// Application/UserCode/MCU/MCU_VAR_1
VAR_GLOBAL
	(********************************************************)
	(*Rx*)
	(*MCUCommandResponse*)
	gu8_MCU_State						:	USINT;
	gu8_MCU_OperationalMode				:	USINT;
	gq_MCU_RegenDeratingStatus			:	BOOL;
	gu8_MCU_RegenDerating				:	USINT;
	gu8_MCU_TractionDerating			:	USINT;
	gu16_MCU_MaxMotorSpeedForward_Rx	:	UINT;
	gu16_MCU_MaxMotorSpeedReverse_Rx	:	UINT;
	gq_MCU_MaxMotorSpeedForwardStatus	:	BOOL;
	gq_MCU_MaxMotorSpeedReverseStatus	:	BOOL;
	gq_MCU_TractionDeratingStatus		:	BOOL;
	gu8_MCU_RollingCounter_Comm1		:	USINT;
	(*MCUCommandResponse2*)
	gu16_MCU_MotorSpeed_Rx				:	UINT;
	gu16_MCU_MotorAngle_Rx				:	UINT;
	gq_MVU_MotorAngleStatus				:	BOOL;
	gq_MCU_MotorSpeedStatus				:	BOOL;
	gq_MCU_SpeedReductionRequest		:	BOOL;
	gq_MCU_EmergencyStop				:	BOOL;
	gu8_MCU_RollingCounter_Comm2		:	USINT;
	(*MCUEventInfo1*)
	gq_MCU_Fault_PhaseToChassis					:	BOOL;
	gq_MCU_Fault_InterlockBatteryCable			:	BOOL;
	gq_MCU_Fault_InterlockMotorCable			:	BOOL;
	gq_MCU_Fault_DriveCoverWasOpened			:	BOOL;
	gq_MCU_Fault_PhaseToChassisStatus			:	BOOL;
	gq_MCU_Fault_InterlockBatteryCableStatus	:	BOOL;
	gq_MCU_Fault_InterlockMotorCableStatus		:	BOOL;
	gq_MCU_Fault_DriveCoverWasOpenedStatus		:	BOOL;
	(*MCUInfo1*)
	gu8_MCU_AuxiliaryVoltage_Rx					:	USINT;
	gu16_MCU_HighPowerVoltage					:	UINT;
	gq_MCU_HighPowerCurrentStatus				:	BOOL;
	gq_MCU_AuxiliaryVoltageStatus				:	BOOL;
	gq_MCU_HighPowerVoltageStatus				:	BOOL;
	gu16_MCU_HighPowerCurrent_Rx				:	UINT;
	gu8_MCU_RollingCounter_Info1				:	USINT;
	(*MCUInfo2*)
	gu16_MCU_MotorTorqueEstimated_Rx			:	UINT;
	gu16_MCU_TractionTorqueAvailable_Rx			:	UINT;
	gu16_MCU_RegenTorqueAvailable_Rx			:	UINT;
	gq_MCU_MotorTorqueEstimatedStatus			:	BOOL;
	gq_MCU_TractionTorqueAvailableStatus		:	BOOL;
	gq_MCU_RegenTorqueAvailableStatus			:	BOOL;
	gu8_MCU_RollingCounter_Info2				:	USINT;
	(*MCUOnEventInfo1*)
	gu16_MCU_EventID							:	UINT;
	gu8_MCU_RollingCounter_OnEventInfo1			:	USINT;
	(*MCUThermal1*)
	gu8_MCU_DriveCoolingFlowRequest_Rx			:	USINT;
	gu8_MCU_MotorCoolingFlowRequest_Rx			:	USINT;
	gu8_MCU_ThermalIndicator_Rx					:	USINT;
	gq_MCU_DriveCoolingFlowRequestStatus		:	BOOL;
	gq_MCU_MotorCoolingFlowRequestStatus		:	BOOL;
	gq_MCU_ThermalIndicatorStatus				:	BOOL;
	gu8_MCU_RollingCounter_Thermal1				:	USINT;
	(*MCUPollingMCUResponse*)
	gq_MCU_ResponseAcknowledgement				:	BOOL;
	gu8_MCU_MCUPollResponse_Multiplex			:	USINT;
		(*MCU MaxMotorSpeed*)
		gu16_MCU_MaxMotorSpeed_Rx				:	UINT;
		(*MCU MaxMotorTorque*)
		gu16_MCU_MaxMotorTorque_Rx				:	UINT;
		(*MCU ProtocolVersion*)
		gu8_MCU_MajorMCUProtocol				:	USINT;
		gu8_MCU_MinorMCUProtocol				:	USINT;
		gu8_MCU_ExtensionMajor					:	USINT;
		gu8_MCU_ExtensionMinor					:	USINT;
		(*MCU SWVersion1*)
		gu8_MCU_MajorMCUSW						:	USINT;
		gu8_MCU_MinorMCUSW						:	USINT;
		gu16_MCU_BranchMCUSW					:	UINT;
		(*MCU SWVersion2*)
		gu32_MCU_RevisionMCUSW					:	UDINT;
		(*MCU TotalMotorRotation*)
		gu32_MCU_TotalMotorRotation_LSB			:	UDINT;
		gu32_MCU_TotalMotorRotation_MSB			:	UDINT;
		gr_MCU_TotalMotorRotation_LSB			:	REAL;
		gr_MCU_TotalMotorRotation_MSB			:	REAL;
		gr_MCU_TotalMotorRotation				:	REAL;
		;
		(*MCUPollingVMU*)
		gu8_MCU_VMUBootNumber						:	USINT;
		(*VMUBootNumber*)
		gu16_MCU_BootNumber						:	UINT;
	
	(***************************************************************)
	(*Rx Conversion*)
	gr_MCU_MaxMotorSpeedForward		:	REAL;
	gr_MCU_MaxMotorSpeedReverse		:	REAL;
	gr_MCU_MotorSpeed				:	REAL;
	gr_MCU_MotorAngle				:	REAL;
	gr_MCU_AuxiliaryVoltage			:	REAL;
	gr_MCU_HighPowerCurrent			:	REAL;
	gr_MCU_MotorTorqueEstimated		:	REAL;
	gr_MCU_TractionTorqueAvailable	:	REAL;
	gr_MCU_RegenTorqueAvailable		:	REAL;
	gr_MCU_DriveCoolingFlowRequest	:	REAL;
	gr_MCU_MotorCoolingFlowRequest	:	REAL;
	gr_MCU_ThermalIndicator			:	REAL;
	gr_MCU_MaxMotorSpeed			:	REAL;
	gr_MCU_MaxMotorTorque			:	REAL;
	(****************************************************************)
	(*Tx*)
	(*VMU Comm1*)
	gu16_MCU_MaxChargeCurrent		:	UINT;
	gu8_MCU_OperationRequest		:	USINT;
	gu16_MCU_MaxDischargeCurrent	:	UINT;
	gu16_MCU_MaxBatteryVoltage		:	UINT;
	gq_MCU_MaxDiscahrgeCurrentStatus	:	BOOL;
	gq_MCU_MaxBatteryVoltageStatus	:	BOOL;
	gq_MCU_MinBatteryVoltageStatus	:	BOOL;
	gq_MCU_MaxChargeCurrentStatus	:	BOOL;
	gu16_MCU_MinBatteryVoltage		:	UINT;
	gu8_MCU_RollingCounter_VMUComm1	:	USINT;
	(*VMU Comm2*)
	gu8_MCU_OperationalMode_Tx		:	USINT;
	gu8_MCU_CommandMode				:	USINT;
	gq_MCU_SpeedCommandStatus		:	BOOL;
	gq_MCU_TorqueCommandStatus		:	BOOL;
	gu16_MCU_TorqueCommand_Tx		:	UINT;
	gu16_MCU_SpeedCommand_Tx		:	UINT;
	gu8_MCU_RollingCounter_VMUComm2	:	USINT;
	(*VMU CommandSafety*)
	gu16_MCU_ReferenceTorqueCommand_Tx	:	UINT;
	gu16_MCU_ReferenceSpeedCommand_Tx	:	UINT;
	gu8_MCU_ReferenceCommandMode		:	USINT;
	gu8_MCU_RollingCounter_VMUCommSafety	:	USINT;
	(*VMUPollingMCU*)
	gu8_MCU_VMUPollMCU_Multiplex	:	USINT;
		(*MCUMaxMotorSpeed*)
		gu16_MCU_MaxMotorSpeed_Tx	:	UINT;
		(*MCUMaxMotorTorque*)
		gu16_MCU_MaxMotorTorque_Tx	:	UINT;
		(*MCUProtocolVersion*)
		gu8_MCU_MajorMCUProtocol_Tx	:	USINT;
		gu8_MCU_MinorMCUProtocol_Tx	:	USINT;
		(*MCUSWVersion1*)
		gu8_MCU_MajorMCUSW_Tx			:	USINT;
		gu8_MCU_MinorMCUSW_Tx			:	USINT;
		gu16_MCU_BranchMCUSW_Tx			:	UINT;
		(*MCUSWVersion2*)
		gu32_MCU_RevisionMCUSW_Tx		:	UDINT;
		(*MCUTotalMotorRotation*)
		gu32_MCU_TotalMotorRotation_LSB_Tx	:	UDINT;
		gu32_MCU_TotalMotorRotation_MSB_Tx	:	UDINT;
	(*VMUPollingVMUResponse*)
	gq_MCU_PollVMUResponse_Acknowledgement	:	BOOL;
	gu8_MCU_PollVMUResponse_Multiplex		:	USINT;
		(*BootNumber*)
		gu16_MCU_BootNumber_Tx			:	UINT;		
	(*VMUSelectProtocolVersion*)
	gu8_MCU_SelectMajorMCUProtocol_Tx		:	USINT;
	gu8_MCU_SelectMinorMCUProtocol_Tx		:	USINT;
	
	(****************************************************************)
	(*True values - pre Tx*)
	gr_MCU_TorqueCommand_PreCF			:	REAL;
	gr_MCU_TorqueCommand_PreCF_Limited	:	REAL;
	gr_MCU_SpeedCommand_PreCF			:	REAL;
	gr_MCU_ReferenceTorqueCommand_PreCF	:	REAL;
	gr_MCU_ReferenceSpeedCommand_PreCF	:	REAL;
	gr_MCU_MaxMotorSpeed_PreCF			:	REAL;
	
	(****************************************************************)
	(*Latching Gear Selection*)
	gq_Gear_Neutral						:	BOOL;
	gq_Gear_Drive						:	BOOL;
	gq_Gear_DriveCrawl					:	BOOL;
	gq_Gear_Reverse						:	BOOL;
	gq_Gear_ReverseCrawl				:	BOOL;
	
	gq_MCU_CommsLoss					:	BOOL;
	
	(*Drivability*)
	gq_ABS_TorqueDisable				:	BOOL;
	
	gr_RearAxle_RelativeSpeed_kph		:	REAL;
	gu8_TractionLoss					:	USINT;
	gr_LeftWheels_RelativeSpeed_kph		:	REAL;
	gr_RightWheels_RelativeSpeed_kph	:	REAL;
	gu8_StabilityLoss					:	USINT;
	gq_ZeroTorqueRq						:	BOOL;
	gton_TorqueReIntro_Timer			:	TON;
	
	gr_RegenSOCMultiplier				:	REAL;
	gr_RegenMultiplierRq				:	REAL;
	gr_RegenIntroCF						:	REAL;
	gq_RegenActive						:	BOOL;
	gr_RegenSpeedDegrading				:	REAL;
	
	
	gr_VehicleTripDistance				:	REAL;
	gr_VehicleInitialTripDistance		:	REAL;
	
	gr_TorqueReIntro					:	REAL;
	gr_TorqueReIntroMax					:	REAL;
	
	gr_MCU_TorqueCommand_Limited	:	REAL;
	gr_MCU_PreviousTorqueCommand	:	REAL;
	
	gq_InitialProtocolGrab			:	BOOL;
END_VAR
VAR_GLOBAL CONSTANT
	MAXMOTORSPEED				:	USINT	:=	2;
	MAXMOTORTORQUE				:	USINT	:=	1;
	PROTOCOLVERSION				:	USINT	:=	0;
	SWVERSION1					:	USINT	:=	3;
	SWVERSION2					:	USINT	:=	4;
	TOTALMOTORROTATION			:	USINT	:=	5;
	TOTALMOTORROTATIONUSINTMCU	:	USINT	:=	6;
	
	VMUBOOTNUMBER				:	USINT	:=	0;
END_VAR

// Application/UserCode/Sevcon_Compressor/Sevcon2_VAR
VAR_GLOBAL
	(*********************************************************)
	
	(*Transmit*)
	(*Torque Demands 1*)
	gu16_Sevcon2_TorqueRq_Tx				:	UINT;
	gu16_Sevcon2_Controlword				:	UINT;
	gu16_Sevcon2_TorqueTractionLimit_Tx		:	UINT;
	gu8_Sevcon2_SEQCommand1					:	USINT;
	gu8_Sevcon2_CSCommand1					:	USINT;
	
	(*Torque Demands 2*)
	gu16_Sevcon2_TorqueRegenLimit_Tx		:	UINT;
	gu16_Sevcon2_SpeedLimitForward			:	UINT;
	gs16_Sevcon2_SpeedLimitReverse			:	INT;
	gu8_Sevcon2_SEQCommand2					:	USINT;
	gu8_Sevcon2_CSCommand2					:	USINT;
	
	(*Battery Demands*)
	gu16_Sevcon2_DCLink_ImaxDischarge		:	UINT;
	gs16_Sevcon2_DCLink_ImaxRecharge		:	INT;
	gu16_Sevcon2_DCLink_VoltageTarget_Tx	:	UINT;
	gu8_Sevcon2_SEQCurrentLimits			:	USINT;
	gu8_Sevcon2_CSCurrentLimits				:	USINT;
	
	(*I Demand Control*)
	gu16_Sevcon2_DebugIqDirectControl_Tx	:	UINT;
	gu16_Sevcon2_DebugIdDirectControl_Tx	:	UINT;
	gu8_Sevcon2_DirectCurrents				:	USINT;
	gu8_Sevcon2_CSDirectCurrents			:	USINT;
	
	(*********************************************************)
	
	(*Receive*)
	(*Torque Status 1*)
	gs16_Sevcon2_TorqueMeasured_Rx		:	INT;
	gs16_Sevcon2_SpeedMeasured			:	INT;
	gs16_Sevcon2_DCLink_Current			:	INT;
	gu8_Sevcon2_SEQ_Torque				:	USINT;
	gu8_Sevcon2_CS_Torque				:	USINT;
	
	(*Torque Status 2*)
	gs16_Sevcon2_TorqueAvailableForward_Rx	:	INT;
	gs16_Sevcon2_TorqueAvailableReverse_Rx	:	INT;
	gu8_Sevcon2_InverterStatus			:	USINT;
	gu8_Sevcon2_TorqueLimitCode			:	USINT;
	gu8_Sevcon2_SEQ_Status				:	USINT;
	gu8_Sevcon2_CS_Status				:	USINT;
	
	(*Temperature*)
	gs16_Sevcon2_TempRemaining			:	INT;
	gs16_Sevcon2_MotorTemp				:	INT;
	gs16_Sevcon2_DCLink_Voltage_Rx		:	INT;
	gu8_Sevcon2_SEQ_Temp					:	USINT;
	gu8_Sevcon2_CS_Temp					:	USINT;
	
	(**)
	gs16_Sevcon2_FaultCode				:	INT;
	gs32_Sevcon2_FaultData				:	DINT;
	gu8_Sevcon2_SEQ_Fault				:	USINT;
	gu8_Sevcon2_CS_Fault					:	USINT;
	
	(**)
	gs32_Sevcon2_EncoderPosition_Rx		:	DINT;
	
	(**)
	gs16_Sevcon2_Debug_Id_Act_Rx			:	INT;
	gs16_Sevcon2_Debug_Iq_Act_Rx			:	INT;
	gs16_Sevcon2_Debug_Id_Ref_Rx			:	INT;
	gs16_Sevcon2_Debug_Iq_Ref_Rx			:	INT;
	
	(**)
	gu8_Sevcon2_Debug_Temp_Junction0		:	USINT;
	gu8_Sevcon2_Debug_Temp_Junction1		:	USINT;
	gu8_Sevcon2_Debug_Temp_Junction2		:	USINT;
	gu8_Sevcon2_Debug_Temp_Junction3		:	USINT;
	gu8_Sevcon2_Debug_Temp_Junction4		:	USINT;
	gu8_Sevcon2_Debug_Temp_Junction5		:	USINT;
	gu8_Sevcon2_Debug_Temp_MotorMeasured	:	USINT;
	gu8_Sevcon2_Debug_Temp_MotorEstimate	:	USINT;
	
	(**)
	gu8_Sevcon2_Debug_Temp_CapEstimateFast	:	USINT;
	gu8_Sevcon2_Debug_Temp_Track				:	USINT;
	gu8_Sevcon2_Debug_Temp_CapEstimateSlow	:	USINT;
	gu8_Sevcon2_Debug_Temp_Heatsink			:	USINT;
	gu8_Sevcon2_Debug_Temp_DeltaTj			:	USINT;
	gu8_Sevcon2_Debug_Temp_Normalised		:	USINT;
	gu8_Sevcon2_Debug_Temp_Coolant			:	USINT;
	gu8_Sevcon2_Debug_Temp_Winding			:	USINT;
	
	(**)
	gs16_Sevcon2_Debug_MaxFlux				:	INT;
	gs16_Sevcon2_Debug_IvLim					:	INT;
	gs16_Sevcon2_Debug_IqMax					:	INT;
	gs16_Sevcon2_Debug_Ls_Rx					:	INT;
	
	(**)
	gs16_Sevcon2_Debug_Slip_Rx				:	INT;
	gs16_Sevcon2_Debug_LmSat_Rx				:	INT;
	gs16_Sevcon2_Debug_IqMax2				:	INT;
	gs16_Sevcon2_Debug_RecipFlux				:	INT;
	
	(*********************************************************)
	(*Tx conversion*)
	gr_Sevcon2_TorqueRq					:	REAL;
	gr_Sevcon2_TorqueTractionLimit		:	REAL;
	gr_Sevcon2_TorqueRegenLimit			:	REAL;
	gr_Sevcon2_DCLink_VoltageTarget		:	REAL;
	gr_Sevcon2_DebugIqDirectControl		:	REAL;
	gr_Sevcon2_DebugIdDirectControl		:	REAL;
	
	(*********************************************************)
	(*Rx converison*)
	gr_Sevcon2_TorqueMeasured			:	REAL;
	gr_Sevcon2_TorqueAvailableForward	:	REAL;
	gr_Sevcon2_TorqueAvailableReverse	:	REAL;
	gr_Sevcon2_DCLink_Voltage			:	REAL;
	gr_Sevcon2_EncoderPosition			:	REAL;
	gr_Sevcon2_Debug_Id_Act				:	REAL;
	gr_Sevcon2_Debug_Iq_Act				:	REAL;
	gr_Sevcon2_Debug_Id_Ref				:	REAL;
	gr_Sevcon2_Debug_Iq_Ref				:	REAL;
	gr_Sevcon2_Debug_Ls					:	REAL;
	gr_Sevcon2_Debug_Slip				:	REAL;
	gr_Sevcon2_Debug_LmSat				:	REAL;
	
	
	gq_Sevcon2_CommsLoss				:	BOOL;
	
END_VAR

// Application/UserCode/Sevcon_Compressor/Sevcon2_VAR_1
VAR_GLOBAL
	(*********************************************************)
	
	(*Transmit*)
	(*Torque Demands 1*)
	gu16_Sevcon2_TorqueRq_Tx				:	UINT;
	gu16_Sevcon2_Controlword				:	UINT;
	gu16_Sevcon2_TorqueTractionLimit_Tx		:	UINT;
	gu8_Sevcon2_SEQCommand1					:	USINT;
	gu8_Sevcon2_CSCommand1					:	USINT;
	
	(*Torque Demands 2*)
	gu16_Sevcon2_TorqueRegenLimit_Tx		:	UINT;
	gu16_Sevcon2_SpeedLimitForward			:	UINT;
	gs16_Sevcon2_SpeedLimitReverse			:	INT;
	gu8_Sevcon2_SEQCommand2					:	USINT;
	gu8_Sevcon2_CSCommand2					:	USINT;
	
	(*Battery Demands*)
	gu16_Sevcon2_DCLink_ImaxDischarge		:	UINT;
	gs16_Sevcon2_DCLink_ImaxRecharge		:	INT;
	gu16_Sevcon2_DCLink_VoltageTarget_Tx	:	UINT;
	gu8_Sevcon2_SEQCurrentLimits			:	USINT;
	gu8_Sevcon2_CSCurrentLimits				:	USINT;
	
	(*I Demand Control*)
	gu16_Sevcon2_DebugIqDirectControl_Tx	:	UINT;
	gu16_Sevcon2_DebugIdDirectControl_Tx	:	UINT;
	gu8_Sevcon2_DirectCurrents				:	USINT;
	gu8_Sevcon2_CSDirectCurrents			:	USINT;
	
	(*********************************************************)
	
	(*Receive*)
	(*Torque Status 1*)
	gs16_Sevcon2_TorqueMeasured_Rx		:	INT;
	gs16_Sevcon2_SpeedMeasured			:	INT;
	gs16_Sevcon2_DCLink_Current			:	INT;
	gu8_Sevcon2_SEQ_Torque				:	USINT;
	gu8_Sevcon2_CS_Torque				:	USINT;
	
	(*Torque Status 2*)
	gs16_Sevcon2_TorqueAvailableForward_Rx	:	INT;
	gs16_Sevcon2_TorqueAvailableReverse_Rx	:	INT;
	gu8_Sevcon2_InverterStatus			:	USINT;
	gu8_Sevcon2_TorqueLimitCode			:	USINT;
	gu8_Sevcon2_SEQ_Status				:	USINT;
	gu8_Sevcon2_CS_Status				:	USINT;
	
	(*Temperature*)
	gs16_Sevcon2_TempRemaining			:	INT;
	gs16_Sevcon2_MotorTemp				:	INT;
	gs16_Sevcon2_DCLink_Voltage_Rx		:	INT;
	gu8_Sevcon2_SEQ_Temp					:	USINT;
	gu8_Sevcon2_CS_Temp					:	USINT;
	
	(**)
	gs16_Sevcon2_FaultCode				:	INT;
	gs32_Sevcon2_FaultData				:	DINT;
	gu8_Sevcon2_SEQ_Fault				:	USINT;
	gu8_Sevcon2_CS_Fault					:	USINT;
	
	(**)
	gs32_Sevcon2_EncoderPosition_Rx		:	DINT;
	
	(**)
	gs16_Sevcon2_Debug_Id_Act_Rx			:	INT;
	gs16_Sevcon2_Debug_Iq_Act_Rx			:	INT;
	gs16_Sevcon2_Debug_Id_Ref_Rx			:	INT;
	gs16_Sevcon2_Debug_Iq_Ref_Rx			:	INT;
	
	(**)
	gu8_Sevcon2_Debug_Temp_Junction0		:	USINT;
	gu8_Sevcon2_Debug_Temp_Junction1		:	USINT;
	gu8_Sevcon2_Debug_Temp_Junction2		:	USINT;
	gu8_Sevcon2_Debug_Temp_Junction3		:	USINT;
	gu8_Sevcon2_Debug_Temp_Junction4		:	USINT;
	gu8_Sevcon2_Debug_Temp_Junction5		:	USINT;
	gu8_Sevcon2_Debug_Temp_MotorMeasured	:	USINT;
	gu8_Sevcon2_Debug_Temp_MotorEstimate	:	USINT;
	
	(**)
	gu8_Sevcon2_Debug_Temp_CapEstimateFast	:	USINT;
	gu8_Sevcon2_Debug_Temp_Track				:	USINT;
	gu8_Sevcon2_Debug_Temp_CapEstimateSlow	:	USINT;
	gu8_Sevcon2_Debug_Temp_Heatsink			:	USINT;
	gu8_Sevcon2_Debug_Temp_DeltaTj			:	USINT;
	gu8_Sevcon2_Debug_Temp_Normalised		:	USINT;
	gu8_Sevcon2_Debug_Temp_Coolant			:	USINT;
	gu8_Sevcon2_Debug_Temp_Winding			:	USINT;
	
	(**)
	gs16_Sevcon2_Debug_MaxFlux				:	INT;
	gs16_Sevcon2_Debug_IvLim					:	INT;
	gs16_Sevcon2_Debug_IqMax					:	INT;
	gs16_Sevcon2_Debug_Ls_Rx					:	INT;
	
	(**)
	gs16_Sevcon2_Debug_Slip_Rx				:	INT;
	gs16_Sevcon2_Debug_LmSat_Rx				:	INT;
	gs16_Sevcon2_Debug_IqMax2				:	INT;
	gs16_Sevcon2_Debug_RecipFlux				:	INT;
	
	(*********************************************************)
	(*Tx conversion*)
	gr_Sevcon2_TorqueRq					:	REAL;
	gr_Sevcon2_TorqueTractionLimit		:	REAL;
	gr_Sevcon2_TorqueRegenLimit			:	REAL;
	gr_Sevcon2_DCLink_VoltageTarget		:	REAL;
	gr_Sevcon2_DebugIqDirectControl		:	REAL;
	gr_Sevcon2_DebugIdDirectControl		:	REAL;
	
	(*********************************************************)
	(*Rx converison*)
	gr_Sevcon2_TorqueMeasured			:	REAL;
	gr_Sevcon2_TorqueAvailableForward	:	REAL;
	gr_Sevcon2_TorqueAvailableReverse	:	REAL;
	gr_Sevcon2_DCLink_Voltage			:	REAL;
	gr_Sevcon2_EncoderPosition			:	REAL;
	gr_Sevcon2_Debug_Id_Act				:	REAL;
	gr_Sevcon2_Debug_Iq_Act				:	REAL;
	gr_Sevcon2_Debug_Id_Ref				:	REAL;
	gr_Sevcon2_Debug_Iq_Ref				:	REAL;
	gr_Sevcon2_Debug_Ls					:	REAL;
	gr_Sevcon2_Debug_Slip				:	REAL;
	gr_Sevcon2_Debug_LmSat				:	REAL;
	
	
	gq_Sevcon2_CommsLoss				:	BOOL;
	
END_VAR

// Application/UserCode/Sevcon ePTO/Sevcon_ePTO_VAR
VAR_GLOBAL
	(*********************************************************)
	
	(*Transmit*)
	(*Torque Demands 1*)
	gu16_Sevcon_ePTO_TorqueRq_Tx				:	UINT;
	gu16_Sevcon_ePTO_Controlword				:	UINT;
	gu16_Sevcon_ePTO_TorqueTractionLimit_Tx		:	UINT;
	gu8_Sevcon_ePTO_SEQCommand1					:	USINT;
	gu8_Sevcon_ePTO_CSCommand1					:	USINT;
	
	(*Torque Demands 2*)
	gu16_Sevcon_ePTO_TorqueRegenLimit_Tx		:	UINT;
	gu16_Sevcon_ePTO_SpeedLimitForward			:	UINT;
	gs16_Sevcon_ePTO_SpeedLimitReverse			:	INT;
	gu8_Sevcon_ePTO_SEQCommand2					:	USINT;
	gu8_Sevcon_ePTO_CSCommand2					:	USINT;
	
	(*Battery Demands*)
	gu16_Sevcon_ePTO_DCLink_ImaxDischarge		:	UINT;
	gs16_Sevcon_ePTO_DCLink_ImaxRecharge		:	INT;
	gu16_Sevcon_ePTO_DCLink_VoltageTarget_Tx	:	UINT;
	gu8_Sevcon_ePTO_SEQCurrentLimits			:	USINT;
	gu8_Sevcon_ePTO_CSCurrentLimits				:	USINT;
	
	(*I Demand Control*)
	gu16_Sevcon_ePTO_DebugIqDirectControl_Tx	:	UINT;
	gu16_Sevcon_ePTO_DebugIdDirectControl_Tx	:	UINT;
	gu8_Sevcon_ePTO_DirectCurrents				:	USINT;
	gu8_Sevcon_ePTO_CSDirectCurrents			:	USINT;
	
	(*********************************************************)
	
	(*Receive*)
	(*Torque Status 1*)
	gs16_Sevcon_ePTO_TorqueMeasured_Rx		:	INT;
	gs16_Sevcon_ePTO_SpeedMeasured			:	INT;
	gs16_Sevcon_ePTO_DCLink_Current			:	INT;
	gu8_Sevcon_ePTO_SEQ_Torque				:	USINT;
	gu8_Sevcon_ePTO_CS_Torque				:	USINT;
	
	(*Torque Status 2*)
	gs16_Sevcon_ePTO_TorqueAvailableForward_Rx	:	INT;
	gs16_Sevcon_ePTO_TorqueAvailableReverse_Rx	:	INT;
	gu8_Sevcon_ePTO_InverterStatus			:	USINT;
	gu8_Sevcon_ePTO_TorqueLimitCode			:	USINT;
	gu8_Sevcon_ePTO_SEQ_Status				:	USINT;
	gu8_Sevcon_ePTO_CS_Status				:	USINT;
	
	(*Temperature*)
	gs16_Sevcon_ePTO_TempRemaining			:	INT;
	gs16_Sevcon_ePTO_MotorTemp				:	INT;
	gs16_Sevcon_ePTO_DCLink_Voltage_Rx		:	INT;
	gu8_Sevcon_ePTO_SEQ_Temp					:	USINT;
	gu8_Sevcon_ePTO_CS_Temp					:	USINT;
	
	(**)
	gs16_Sevcon_ePTO_FaultCode				:	INT;
	gs32_Sevcon_ePTO_FaultData				:	DINT;
	gu8_Sevcon_ePTO_SEQ_Fault				:	USINT;
	gu8_Sevcon_ePTO_CS_Fault					:	USINT;
	
	(**)
	gs32_Sevcon_ePTO_EncoderPosition_Rx		:	DINT;
	
	(**)
	gs16_Sevcon_ePTO_Debug_Id_Act_Rx			:	INT;
	gs16_Sevcon_ePTO_Debug_Iq_Act_Rx			:	INT;
	gs16_Sevcon_ePTO_Debug_Id_Ref_Rx			:	INT;
	gs16_Sevcon_ePTO_Debug_Iq_Ref_Rx			:	INT;
	
	(**)
	gu8_Sevcon_ePTO_Debug_Temp_Junction0		:	USINT;
	gu8_Sevcon_ePTO_Debug_Temp_Junction1		:	USINT;
	gu8_Sevcon_ePTO_Debug_Temp_Junction2		:	USINT;
	gu8_Sevcon_ePTO_Debug_Temp_Junction3		:	USINT;
	gu8_Sevcon_ePTO_Debug_Temp_Junction4		:	USINT;
	gu8_Sevcon_ePTO_Debug_Temp_Junction5		:	USINT;
	gu8_Sevcon_ePTO_Debug_Temp_MotorMeasured	:	USINT;
	gu8_Sevcon_ePTO_Debug_Temp_MotorEstimate	:	USINT;
	
	(**)
	gu8_Sevcon_ePTO_Debug_Temp_CapEstimateFast	:	USINT;
	gu8_Sevcon_ePTO_Debug_Temp_Track				:	USINT;
	gu8_Sevcon_ePTO_Debug_Temp_CapEstimateSlow	:	USINT;
	gu8_Sevcon_ePTO_Debug_Temp_Heatsink			:	USINT;
	gu8_Sevcon_ePTO_Debug_Temp_DeltaTj			:	USINT;
	gu8_Sevcon_ePTO_Debug_Temp_Normalised		:	USINT;
	gu8_Sevcon_ePTO_Debug_Temp_Coolant			:	USINT;
	gu8_Sevcon_ePTO_Debug_Temp_Winding			:	USINT;
	
	(**)
	gs16_Sevcon_ePTO_Debug_MaxFlux				:	INT;
	gs16_Sevcon_ePTO_Debug_IvLim					:	INT;
	gs16_Sevcon_ePTO_Debug_IqMax					:	INT;
	gs16_Sevcon_ePTO_Debug_Ls_Rx					:	INT;
	
	(**)
	gs16_Sevcon_ePTO_Debug_Slip_Rx				:	INT;
	gs16_Sevcon_ePTO_Debug_LmSat_Rx				:	INT;
	gs16_Sevcon_ePTO_Debug_IqMax2				:	INT;
	gs16_Sevcon_ePTO_Debug_RecipFlux				:	INT;
	
	(*********************************************************)
	(*Tx conversion*)
	gr_Sevcon_ePTO_TorqueRq					:	REAL;
	gr_Sevcon_ePTO_TorqueTractionLimit		:	REAL;
	gr_Sevcon_ePTO_TorqueRegenLimit			:	REAL;
	gr_Sevcon_ePTO_DCLink_VoltageTarget		:	REAL;
	gr_Sevcon_ePTO_DebugIqDirectControl		:	REAL;
	gr_Sevcon_ePTO_DebugIdDirectControl		:	REAL;
	
	(*********************************************************)
	(*Rx converison*)
	gr_Sevcon_ePTO_TorqueMeasured			:	REAL;
	gr_Sevcon_ePTO_TorqueAvailableForward	:	REAL;
	gr_Sevcon_ePTO_TorqueAvailableReverse	:	REAL;
	gr_Sevcon_ePTO_DCLink_Voltage			:	REAL;
	gr_Sevcon_ePTO_EncoderPosition			:	REAL;
	gr_Sevcon_ePTO_Debug_Id_Act				:	REAL;
	gr_Sevcon_ePTO_Debug_Iq_Act				:	REAL;
	gr_Sevcon_ePTO_Debug_Id_Ref				:	REAL;
	gr_Sevcon_ePTO_Debug_Iq_Ref				:	REAL;
	gr_Sevcon_ePTO_Debug_Ls					:	REAL;
	gr_Sevcon_ePTO_Debug_Slip				:	REAL;
	gr_Sevcon_ePTO_Debug_LmSat				:	REAL;
	
	
	
	
END_VAR

// Application/UserCode/Sevcon_PSP/Sevcon_Steer_VAR_1
VAR_GLOBAL
	(*********************************************************)
	
	(*Transmit*)
	(*Torque Demands 1*)
	gu16_Sevcon1_TorqueRq_Tx				:	UINT;
	gu16_Sevcon1_Controlword				:	UINT;
	gu16_Sevcon1_TorqueTractionLimit_Tx		:	UINT;
	gu8_Sevcon1_SEQCommand1					:	USINT;
	gu8_Sevcon1_CSCommand1					:	USINT;
	
	(*Torque Demands 2*)
	gu16_Sevcon1_TorqueRegenLimit_Tx		:	UINT;
	gu16_Sevcon1_SpeedLimitForward			:	UINT;
	gs16_Sevcon1_SpeedLimitReverse			:	INT;
	gu8_Sevcon1_SEQCommand2					:	USINT;
	gu8_Sevcon1_CSCommand2					:	USINT;
	
	(*Battery Demands*)
	gu16_Sevcon1_DCLink_ImaxDischarge		:	UINT;
	gs16_Sevcon1_DCLink_ImaxRecharge		:	INT;
	gu16_Sevcon1_DCLink_VoltageTarget_Tx	:	UINT;
	gu8_Sevcon1_SEQCurrentLimits			:	USINT;
	gu8_Sevcon1_CSCurrentLimits				:	USINT;
	
	(*I Demand Control*)
	gu16_Sevcon1_DebugIqDirectControl_Tx	:	UINT;
	gu16_Sevcon1_DebugIdDirectControl_Tx	:	UINT;
	gu8_Sevcon1_DirectCurrents				:	USINT;
	gu8_Sevcon1_CSDirectCurrents			:	USINT;
	
	(*********************************************************)
	
	(*Receive*)
	(*Torque Status 1*)
	gs16_Sevcon1_TorqueMeasured_Rx		:	INT;
	gs16_Sevcon1_SpeedMeasured			:	INT;
	gs16_Sevcon1_DCLink_Current			:	INT;
	gu8_Sevcon1_SEQ_Torque				:	USINT;
	gu8_Sevcon1_CS_Torque				:	USINT;
	
	(*Torque Status 2*)
	gs16_Sevcon1_TorqueAvailableForward_Rx	:	INT;
	gs16_Sevcon1_TorqueAvailableReverse_Rx	:	INT;
	gu8_Sevcon1_InverterStatus			:	USINT;
	gu8_Sevcon1_TorqueLimitCode			:	USINT;
	gu8_Sevcon1_SEQ_Status				:	USINT;
	gu8_Sevcon1_CS_Status				:	USINT;
	
	(*Temperature*)
	gs16_Sevcon1_TempRemaining			:	INT;
	gs16_Sevcon1_MotorTemp				:	INT;
	gs16_Sevcon1_DCLink_Voltage_Rx		:	INT;
	gu8_Sevcon1_SEQ_Temp					:	USINT;
	gu8_Sevcon1_CS_Temp					:	USINT;
	
	(**)
	gs16_Sevcon1_FaultCode				:	INT;
	gs32_Sevcon1_FaultData				:	DINT;
	gu8_Sevcon1_SEQ_Fault				:	USINT;
	gu8_Sevcon1_CS_Fault					:	USINT;
	
	(**)
	gs32_Sevcon1_EncoderPosition_Rx		:	DINT;
	
	(**)
	gs16_Sevcon1_Debug_Id_Act_Rx			:	INT;
	gs16_Sevcon1_Debug_Iq_Act_Rx			:	INT;
	gs16_Sevcon1_Debug_Id_Ref_Rx			:	INT;
	gs16_Sevcon1_Debug_Iq_Ref_Rx			:	INT;
	
	(**)
	gu8_Sevcon1_Debug_Temp_Junction0		:	USINT;
	gu8_Sevcon1_Debug_Temp_Junction1		:	USINT;
	gu8_Sevcon1_Debug_Temp_Junction2		:	USINT;
	gu8_Sevcon1_Debug_Temp_Junction3		:	USINT;
	gu8_Sevcon1_Debug_Temp_Junction4		:	USINT;
	gu8_Sevcon1_Debug_Temp_Junction5		:	USINT;
	gu8_Sevcon1_Debug_Temp_MotorMeasured	:	USINT;
	gu8_Sevcon1_Debug_Temp_MotorEstimate	:	USINT;
	
	(**)
	gu8_Sevcon1_Debug_Temp_CapEstimateFast	:	USINT;
	gu8_Sevcon1_Debug_Temp_Track				:	USINT;
	gu8_Sevcon1_Debug_Temp_CapEstimateSlow	:	USINT;
	gu8_Sevcon1_Debug_Temp_Heatsink			:	USINT;
	gu8_Sevcon1_Debug_Temp_DeltaTj			:	USINT;
	gu8_Sevcon1_Debug_Temp_Normalised		:	USINT;
	gu8_Sevcon1_Debug_Temp_Coolant			:	USINT;
	gu8_Sevcon1_Debug_Temp_Winding			:	USINT;
	
	(**)
	gs16_Sevcon1_Debug_MaxFlux				:	INT;
	gs16_Sevcon1_Debug_IvLim					:	INT;
	gs16_Sevcon1_Debug_IqMax					:	INT;
	gs16_Sevcon1_Debug_Ls_Rx					:	INT;
	
	(**)
	gs16_Sevcon1_Debug_Slip_Rx				:	INT;
	gs16_Sevcon1_Debug_LmSat_Rx				:	INT;
	gs16_Sevcon1_Debug_IqMax2				:	INT;
	gs16_Sevcon1_Debug_RecipFlux				:	INT;
	
	(*********************************************************)
	(*Tx conversion*)
	gr_Sevcon1_TorqueRq					:	REAL;
	gr_Sevcon1_TorqueTractionLimit		:	REAL;
	gr_Sevcon1_TorqueRegenLimit			:	REAL;
	gr_Sevcon1_DCLink_VoltageTarget		:	REAL;
	gr_Sevcon1_DebugIqDirectControl		:	REAL;
	gr_Sevcon1_DebugIdDirectControl		:	REAL;
	
	(*********************************************************)
	(*Rx converison*)
	gr_Sevcon1_TorqueMeasured			:	REAL;
	gr_Sevcon1_TorqueAvailableForward	:	REAL;
	gr_Sevcon1_TorqueAvailableReverse	:	REAL;
	gr_Sevcon1_DCLink_Voltage			:	REAL;
	gr_Sevcon1_EncoderPosition			:	REAL;
	gr_Sevcon1_Debug_Id_Act				:	REAL;
	gr_Sevcon1_Debug_Iq_Act				:	REAL;
	gr_Sevcon1_Debug_Id_Ref				:	REAL;
	gr_Sevcon1_Debug_Iq_Ref				:	REAL;
	gr_Sevcon1_Debug_Ls					:	REAL;
	gr_Sevcon1_Debug_Slip				:	REAL;
	gr_Sevcon1_Debug_LmSat				:	REAL;
	
	
	gq_Sevcon1_CommsLoss				:	BOOL;
	
END_VAR

// Application/UserCode/UserMramUsage_1/UserMramVariables_1
VAR_GLOBAL
	///[Pointer to the start of the NVRAM area.]
	G_pUserMramStructure: POINTER TO UserMramStructure;
	///[Pointer to the start of the OD parameter image.]
	G_UserMramStructureDefault: UserMramStructure;
END_VAR

// Application/UserCode/UserMramUsage/UserMramVariables
VAR_GLOBAL
	///[Pointer to the start of the NVRAM area.]
	G_pUserMramStructure: POINTER TO UserMramStructure;
	///[Pointer to the start of the OD parameter image.]
	G_UserMramStructureDefault: UserMramStructure;
END_VAR

// Application/CodeTemplate/Globals/CANopen_CAN1/G_CAN1_VAR
///
///NOTE! NOTE! NOTE! NOTE! NOTE! NOTE! NOTE! NOTE! NOTE! NOTE! NOTE!
/// 	                    
/// This object is created by Epec MultiTool
/// User changes are overwritten when project is imported
///
/// Content
/// - CANopen OD index data
///
{attribute 'qualified_only'}
VAR_GLOBAL
	/// 16#1000 Information about the device type
	DeviceType_Device1: UDINT := 405;
	/// 16#1001 Error information
	ErrorReg_Device1: USINT := 0;
	/// 16#2128 PDO Dummy Variable Index
	CAN1_TPDO_DUMMY: BYTE := 0;
	/// 16#2129 PDO Dummy Variable Index
	CAN1_RPDO_DUMMY: BYTE := 0;
	/// 16#2131 Parameter CSV unique ID
	Parameter_CSV_unique_ID1: UINT := 16#0000;
END_VAR

// Application/CodeTemplate/Globals/CANopen_CAN1/G_CANopen_CAN1
///
///NOTE! NOTE! NOTE! NOTE! NOTE! NOTE! NOTE! NOTE! NOTE! NOTE! NOTE!
/// 	                    
/// This object is created by Epec MultiTool
/// User changes are overwritten when project is imported
///
/// Content
/// - CANopen protocol variable definitions
///
{attribute 'qualified_only'}
{attribute 'global_init_slot' := '49991'}
VAR_GLOBAL
	/// CAN device
	Device: EPEC_CANopen.Device;
	/// Object Dictionary data
	OD: EPEC_CANopen.OD;
	ODEntrys: ARRAY[1..74] OF EPEC_CANopen.ODEntry;
	/// Protocol data
	Protocols: ARRAY[1..5] OF EPEC_CANopen.ProtocolEntry;
	/// Heartbeat producer/consumer protocol data
	HB: EPEC_CANopen.HBData;
	/// Heartbeat producer/consumer protocol handler
	HB_Handler: EPEC_CANopen.CANopenHB;
	/// NMT protocol data
	NMT: EPEC_CANopen.NMTData;
	/// NMT protocol handler
	NMT_Handler: EPEC_CANopen.CANopenNMT;
	/// SDO server protocol data
	SSDO: EPEC_CANopen.SSDOData;
	/// SDO server protocol handler
	SSDO_Handler: EPEC_CANopen.CANopenSDOServer;
	/// GFC protocol data
	GFC: EPEC_CANopen.GFCData;
	/// GFC protocol handler
	GFC_Handler: EPEC_CANopen.CANopenGFC;
	/// SDO client instances
	CSDOS: ARRAY[1..127] OF EPEC_CANopen.CANopenCSDO := [];
	SaveAll: EPEC_ODSave.SaveODSaveAll;
	DeleteAll: EPEC_ODSave.SaveODDeleteAll;
	Initialize: EPEC_ODSave.SaveODInitialize;
	SaveData: ARRAY[0..3] OF EPEC_ODSave.SaveODSubIndexDescription := [(StartIndex := 16#1000, EndIndex := 16#FFFF, GroupNum := 1), (StartIndex := 16#1000, EndIndex := 16#1FFF, GroupNum := 1), (StartIndex := 16#2000, EndIndex := 16#FFFF, GroupNum := 1), (StartIndex := 16#0, EndIndex := 16#0, GroupNum := 1)];
	SaveSubData1010h: EPEC_ODSave.SaveODSubService;
END_VAR

// Application/CodeTemplate/Globals/CANopen_CAN1/G_CANopen_CAN1_VAR
///
///NOTE! NOTE! NOTE! NOTE! NOTE! NOTE! NOTE! NOTE! NOTE! NOTE! NOTE!
/// 	                    
/// This object is created by Epec MultiTool
/// User changes are overwritten when project is imported
///
/// Content
/// - 
/// 
{attribute 'qualified_only'}
{attribute 'global_init_slot' := '49990'}
VAR_GLOBAL
	OD_Error: EPEC_CANopen.Errors := EPEC_CANopen.Errors.NotInitialized;
	ODSave_Error: EPEC_ODSave.SaveODErrors;
	Callback_Error: EPEC_CANopen.Errors := EPEC_CANopen.Errors.NotInitialized;
	ProtocolAdded: ARRAY[1..5] OF BOOL := [5(0)];
	HB_Error: EPEC_CANopen.Errors := EPEC_CANopen.Errors.NotInitialized;
	NMT_Error: EPEC_CANopen.Errors := EPEC_CANopen.Errors.NotInitialized;
	SSDO_Error: EPEC_CANopen.Errors := EPEC_CANopen.Errors.NotInitialized;
	GFC_Error: EPEC_CANopen.Errors := EPEC_CANopen.Errors.NotInitialized;
	/// GFC status
	GFC_Status: BYTE;
	CSDO_Error: EPEC_CANopen.Errors := EPEC_CANopen.Errors.NotInitialized;
	SaveSigns1010: ARRAY[0..3] OF DWORD;
END_VAR

// Application/CodeTemplate/Globals/CANopen_CAN2/G_CAN2_VAR
///
///NOTE! NOTE! NOTE! NOTE! NOTE! NOTE! NOTE! NOTE! NOTE! NOTE! NOTE!
/// 	                    
/// This object is created by Epec MultiTool
/// User changes are overwritten when project is imported
///
/// Content
/// - CANopen OD index data
///
{attribute 'qualified_only'}
VAR_GLOBAL
	/// 16#1000 Information about the device type
	DeviceType_Device2: UDINT := 405;
	/// 16#1001 Error information
	ErrorReg_Device2: USINT := 0;
	/// 16#2128 PDO Dummy Variable Index
	CAN2_TPDO_DUMMY: BYTE := 0;
	/// 16#2129 PDO Dummy Variable Index
	CAN2_RPDO_DUMMY: BYTE := 0;
	/// 16#2131 Parameter CSV unique ID
	Parameter_CSV_unique_ID2: UINT := 16#0000;
END_VAR

// Application/CodeTemplate/Globals/CANopen_CAN2/G_CANopen_CAN2
///
///NOTE! NOTE! NOTE! NOTE! NOTE! NOTE! NOTE! NOTE! NOTE! NOTE! NOTE!
/// 	                    
/// This object is created by Epec MultiTool
/// User changes are overwritten when project is imported
///
/// Content
/// - CANopen protocol variable definitions
///
{attribute 'qualified_only'}
{attribute 'global_init_slot' := '49991'}
VAR_GLOBAL
	/// CAN device
	Device: EPEC_CANopen.Device;
	/// Object Dictionary data
	OD: EPEC_CANopen.OD;
	ODEntrys: ARRAY[1..66] OF EPEC_CANopen.ODEntry;
	/// Protocol data
	Protocols: ARRAY[1..5] OF EPEC_CANopen.ProtocolEntry;
	/// Heartbeat producer/consumer protocol data
	HB: EPEC_CANopen.HBData;
	/// Heartbeat producer/consumer protocol handler
	HB_Handler: EPEC_CANopen.CANopenHB;
	/// NMT protocol data
	NMT: EPEC_CANopen.NMTData;
	/// NMT protocol handler
	NMT_Handler: EPEC_CANopen.CANopenNMT;
	/// SDO server protocol data
	SSDO: EPEC_CANopen.SSDOData;
	/// SDO server protocol handler
	SSDO_Handler: EPEC_CANopen.CANopenSDOServer;
	/// GFC protocol data
	GFC: EPEC_CANopen.GFCData;
	/// GFC protocol handler
	GFC_Handler: EPEC_CANopen.CANopenGFC;
	/// SDO client instances
	CSDOS: ARRAY[1..127] OF EPEC_CANopen.CANopenCSDO := [];
	SaveAll: EPEC_ODSave.SaveODSaveAll;
	DeleteAll: EPEC_ODSave.SaveODDeleteAll;
	Initialize: EPEC_ODSave.SaveODInitialize;
	SaveData: ARRAY[0..3] OF EPEC_ODSave.SaveODSubIndexDescription := [(StartIndex := 16#1000, EndIndex := 16#FFFF, GroupNum := 2), (StartIndex := 16#1000, EndIndex := 16#1FFF, GroupNum := 2), (StartIndex := 16#2000, EndIndex := 16#FFFF, GroupNum := 2), (StartIndex := 16#0, EndIndex := 16#0, GroupNum := 2)];
	SaveSubData1010h: EPEC_ODSave.SaveODSubService;
END_VAR

// Application/CodeTemplate/Globals/CANopen_CAN2/G_CANopen_CAN2_VAR
///
///NOTE! NOTE! NOTE! NOTE! NOTE! NOTE! NOTE! NOTE! NOTE! NOTE! NOTE!
/// 	                    
/// This object is created by Epec MultiTool
/// User changes are overwritten when project is imported
///
/// Content
/// - 
/// 
{attribute 'qualified_only'}
{attribute 'global_init_slot' := '49990'}
VAR_GLOBAL
	OD_Error: EPEC_CANopen.Errors := EPEC_CANopen.Errors.NotInitialized;
	ODSave_Error: EPEC_ODSave.SaveODErrors;
	Callback_Error: EPEC_CANopen.Errors := EPEC_CANopen.Errors.NotInitialized;
	ProtocolAdded: ARRAY[1..5] OF BOOL := [5(0)];
	HB_Error: EPEC_CANopen.Errors := EPEC_CANopen.Errors.NotInitialized;
	NMT_Error: EPEC_CANopen.Errors := EPEC_CANopen.Errors.NotInitialized;
	SSDO_Error: EPEC_CANopen.Errors := EPEC_CANopen.Errors.NotInitialized;
	GFC_Error: EPEC_CANopen.Errors := EPEC_CANopen.Errors.NotInitialized;
	/// GFC status
	GFC_Status: BYTE;
	CSDO_Error: EPEC_CANopen.Errors := EPEC_CANopen.Errors.NotInitialized;
	SaveSigns1010: ARRAY[0..3] OF DWORD;
END_VAR

// Application/CodeTemplate/Globals/CANopen_CAN3/G_CAN3_VAR
///
///NOTE! NOTE! NOTE! NOTE! NOTE! NOTE! NOTE! NOTE! NOTE! NOTE! NOTE!
/// 	                    
/// This object is created by Epec MultiTool
/// User changes are overwritten when project is imported
///
/// Content
/// - CANopen OD index data
///
{attribute 'qualified_only'}
VAR_GLOBAL
	/// 16#1000 Information about the device type
	DeviceType_Device3: UDINT := 405;
	/// 16#1001 Error information
	ErrorReg_Device3: USINT := 0;
	/// 16#2129 PDO Dummy Variable Index
	CAN3_PDO_DUMMY: BYTE := 0;
	/// 16#2131 Parameter CSV unique ID
	Parameter_CSV_unique_ID3: UINT := 16#0000;
END_VAR

// Application/CodeTemplate/Globals/CANopen_CAN3/G_CANopen_CAN3
///
///NOTE! NOTE! NOTE! NOTE! NOTE! NOTE! NOTE! NOTE! NOTE! NOTE! NOTE!
/// 	                    
/// This object is created by Epec MultiTool
/// User changes are overwritten when project is imported
///
/// Content
/// - CANopen protocol variable definitions
///
{attribute 'qualified_only'}
{attribute 'global_init_slot' := '49991'}
VAR_GLOBAL
	/// CAN device
	Device: EPEC_CANopen.Device;
	/// Object Dictionary data
	OD: EPEC_CANopen.OD;
	ODEntrys: ARRAY[1..65] OF EPEC_CANopen.ODEntry;
	/// Protocol data
	Protocols: ARRAY[1..5] OF EPEC_CANopen.ProtocolEntry;
	/// Heartbeat producer/consumer protocol data
	HB: EPEC_CANopen.HBData;
	/// Heartbeat producer/consumer protocol handler
	HB_Handler: EPEC_CANopen.CANopenHB;
	/// NMT protocol data
	NMT: EPEC_CANopen.NMTData;
	/// NMT protocol handler
	NMT_Handler: EPEC_CANopen.CANopenNMT;
	/// SDO server protocol data
	SSDO: EPEC_CANopen.SSDOData;
	/// SDO server protocol handler
	SSDO_Handler: EPEC_CANopen.CANopenSDOServer;
	/// GFC protocol data
	GFC: EPEC_CANopen.GFCData;
	/// GFC protocol handler
	GFC_Handler: EPEC_CANopen.CANopenGFC;
	/// SDO client instances
	CSDOS: ARRAY[1..127] OF EPEC_CANopen.CANopenCSDO := [];
	SaveAll: EPEC_ODSave.SaveODSaveAll;
	DeleteAll: EPEC_ODSave.SaveODDeleteAll;
	Initialize: EPEC_ODSave.SaveODInitialize;
	SaveData: ARRAY[0..3] OF EPEC_ODSave.SaveODSubIndexDescription := [(StartIndex := 16#1000, EndIndex := 16#FFFF, GroupNum := 3), (StartIndex := 16#1000, EndIndex := 16#1FFF, GroupNum := 3), (StartIndex := 16#2000, EndIndex := 16#FFFF, GroupNum := 3), (StartIndex := 16#0, EndIndex := 16#0, GroupNum := 3)];
	SaveSubData1010h: EPEC_ODSave.SaveODSubService;
END_VAR

// Application/CodeTemplate/Globals/CANopen_CAN3/G_CANopen_CAN3_VAR
///
///NOTE! NOTE! NOTE! NOTE! NOTE! NOTE! NOTE! NOTE! NOTE! NOTE! NOTE!
/// 	                    
/// This object is created by Epec MultiTool
/// User changes are overwritten when project is imported
///
/// Content
/// - 
/// 
{attribute 'qualified_only'}
{attribute 'global_init_slot' := '49990'}
VAR_GLOBAL
	OD_Error: EPEC_CANopen.Errors := EPEC_CANopen.Errors.NotInitialized;
	ODSave_Error: EPEC_ODSave.SaveODErrors;
	Callback_Error: EPEC_CANopen.Errors := EPEC_CANopen.Errors.NotInitialized;
	ProtocolAdded: ARRAY[1..5] OF BOOL := [5(0)];
	HB_Error: EPEC_CANopen.Errors := EPEC_CANopen.Errors.NotInitialized;
	NMT_Error: EPEC_CANopen.Errors := EPEC_CANopen.Errors.NotInitialized;
	SSDO_Error: EPEC_CANopen.Errors := EPEC_CANopen.Errors.NotInitialized;
	GFC_Error: EPEC_CANopen.Errors := EPEC_CANopen.Errors.NotInitialized;
	/// GFC status
	GFC_Status: BYTE;
	CSDO_Error: EPEC_CANopen.Errors := EPEC_CANopen.Errors.NotInitialized;
	SaveSigns1010: ARRAY[0..3] OF DWORD;
END_VAR

// Application/CodeTemplate/Globals/CANopen_CAN4/G_CAN4_VAR
///
///NOTE! NOTE! NOTE! NOTE! NOTE! NOTE! NOTE! NOTE! NOTE! NOTE! NOTE!
/// 	                    
/// This object is created by Epec MultiTool
/// User changes are overwritten when project is imported
///
/// Content
/// - CANopen OD index data
///
{attribute 'qualified_only'}
VAR_GLOBAL
	/// 16#1000 Information about the device type
	DeviceType_Device4: UDINT := 405;
	/// 16#1001 Error information
	ErrorReg_Device4: USINT := 0;
	/// 16#2129 PDO Dummy Variable Index
	CAN4_PDO_DUMMY: BYTE := 0;
	/// 16#2131 Parameter CSV unique ID
	Parameter_CSV_unique_ID4: UINT := 16#0000;
END_VAR

// Application/CodeTemplate/Globals/CANopen_CAN4/G_CANopen_CAN4
///
///NOTE! NOTE! NOTE! NOTE! NOTE! NOTE! NOTE! NOTE! NOTE! NOTE! NOTE!
/// 	                    
/// This object is created by Epec MultiTool
/// User changes are overwritten when project is imported
///
/// Content
/// - CANopen protocol variable definitions
///
{attribute 'qualified_only'}
{attribute 'global_init_slot' := '49991'}
VAR_GLOBAL
	/// CAN device
	Device: EPEC_CANopen.Device;
	/// Object Dictionary data
	OD: EPEC_CANopen.OD;
	ODEntrys: ARRAY[1..65] OF EPEC_CANopen.ODEntry;
	/// Protocol data
	Protocols: ARRAY[1..5] OF EPEC_CANopen.ProtocolEntry;
	/// Heartbeat producer/consumer protocol data
	HB: EPEC_CANopen.HBData;
	/// Heartbeat producer/consumer protocol handler
	HB_Handler: EPEC_CANopen.CANopenHB;
	/// NMT protocol data
	NMT: EPEC_CANopen.NMTData;
	/// NMT protocol handler
	NMT_Handler: EPEC_CANopen.CANopenNMT;
	/// SDO server protocol data
	SSDO: EPEC_CANopen.SSDOData;
	/// SDO server protocol handler
	SSDO_Handler: EPEC_CANopen.CANopenSDOServer;
	/// GFC protocol data
	GFC: EPEC_CANopen.GFCData;
	/// GFC protocol handler
	GFC_Handler: EPEC_CANopen.CANopenGFC;
	/// SDO client instances
	CSDOS: ARRAY[1..127] OF EPEC_CANopen.CANopenCSDO := [];
	SaveAll: EPEC_ODSave.SaveODSaveAll;
	DeleteAll: EPEC_ODSave.SaveODDeleteAll;
	Initialize: EPEC_ODSave.SaveODInitialize;
	SaveData: ARRAY[0..3] OF EPEC_ODSave.SaveODSubIndexDescription := [(StartIndex := 16#1000, EndIndex := 16#FFFF, GroupNum := 4), (StartIndex := 16#1000, EndIndex := 16#1FFF, GroupNum := 4), (StartIndex := 16#2000, EndIndex := 16#FFFF, GroupNum := 4), (StartIndex := 16#0, EndIndex := 16#0, GroupNum := 4)];
	SaveSubData1010h: EPEC_ODSave.SaveODSubService;
END_VAR

// Application/CodeTemplate/Globals/CANopen_CAN4/G_CANopen_CAN4_VAR
///
///NOTE! NOTE! NOTE! NOTE! NOTE! NOTE! NOTE! NOTE! NOTE! NOTE! NOTE!
/// 	                    
/// This object is created by Epec MultiTool
/// User changes are overwritten when project is imported
///
/// Content
/// - 
/// 
{attribute 'qualified_only'}
{attribute 'global_init_slot' := '49990'}
VAR_GLOBAL
	OD_Error: EPEC_CANopen.Errors := EPEC_CANopen.Errors.NotInitialized;
	ODSave_Error: EPEC_ODSave.SaveODErrors;
	Callback_Error: EPEC_CANopen.Errors := EPEC_CANopen.Errors.NotInitialized;
	ProtocolAdded: ARRAY[1..5] OF BOOL := [5(0)];
	HB_Error: EPEC_CANopen.Errors := EPEC_CANopen.Errors.NotInitialized;
	NMT_Error: EPEC_CANopen.Errors := EPEC_CANopen.Errors.NotInitialized;
	SSDO_Error: EPEC_CANopen.Errors := EPEC_CANopen.Errors.NotInitialized;
	GFC_Error: EPEC_CANopen.Errors := EPEC_CANopen.Errors.NotInitialized;
	/// GFC status
	GFC_Status: BYTE;
	CSDO_Error: EPEC_CANopen.Errors := EPEC_CANopen.Errors.NotInitialized;
	SaveSigns1010: ARRAY[0..3] OF DWORD;
END_VAR

// Application/UserCode/BMS/OrionBMS/OrionBMS2_VAR
VAR_GLOBAL
	(*Orion BMS2 Variables*)
	(******************************************)
	(*Rx*)
	(*6B0*)
	gs16_OrionBMS2_PackCurrent	:	INT;
	gu16_OrionBMS2_PackVoltage	:	UINT;
	gu8_OrionBMS2_RAW_SOC	:	USINT;
	gu16_OrionBMS2_RelayState	:	UINT;
	gu8_OrionBMS2_Custom_Flag_1	:	USINT;
	(*6B1*)
	gu8_OrionBMS2_Isolation_ADC			:	UINT;
	gu8_OrionBMS2_Shortest_Wave			:	UINT;
	gu16_OrionBMS2_Isolation_Clipping	:	UINT;
	gu16_OrionBMS2_Isolation_Threshold 	: UINT;
	(*6B2*)
	gu16_OrionBMS2_DTC_Flags1		:	UINT;
	gu16_OrionBMS2_DTC_Flags2		:	UINT;
	gu16_OrionBMS2_FailsafeStatus	:	UINT;
	gu16_OrionBMS2_CurrentLimit		:	UINT;
	(*6B3*)
	gu8_OrionBMS2_PackHealth			:	USINT;
	gu16_OrionBMS2_PackCycles			:	UINT;
	gu16_OrionBMS2_PackResistance		:	UINT;
	gu8_OrionBMS2_PopulatedCells		:	USINT;
	gu16_OrionBMS2_MaximumPackVoltage	:	UINT;
	(*6B4*)
	gu8_OrionBMS2_HighTemp				:	USINT;
	gu8_OrionBMS2_LowTemp				:	USINT;
	gu8_OrionBMS2_AverageTemp			:	USINT;
	gu8_OrionBMS2_InternalTemp			:	USINT;
	gu16_OrionBMS2_MinimumPackVoltage	:	UINT;  (*minimumPackvoltage*)
	gu16_OrionBMS2_PackAmphours			:	UINT;
	(*6B5*)
	gu16_OrionBMS2_AverageCellVoltage	:	UINT;
	gu16_OrionBMS2_LowCellVoltage		:	UINT;
	gu16_OrionBMS2_HighCellVoltage		:	UINT;
	gu8_OrionBMS2_LowCellVoltNumber		:	USINT;
	gu8_OrionBMS2_HighCellVoltNumber	:	USINT;
	(*6B6*)
	gu8_OrionBMS2_Low_Intres_ID				:	BYTE;
	gu8_OrionBMS2_High_Intres_ID			:	BYTE;
	gu16_OrionBMS2_Low_Cell_Resistance		:	UINT;
	gu16_OrionBMS2_High_Cell_Resistance		:	UINT;
	gu16_OrionBMS2_Average_Cell_Resistance	: 	UINT;
	
	(*6B7*)
	gu8_OrionBMS2_Low_Thermistor_ID			:	BYTE;
	gu8_OrionBMS2_High_Thermistor_ID		:	BYTE;
	gu16_OrionBMS2_PackDCL					:	UINT;
	gu16_OrionBMS2_PackCCL					:	UINT;
	gu16_OrionBMS2_PackSummedVoltage		:	UINT;
	
	(*6B8*)
	gu8_OrionBMS2_Firmware_Minor			:BYTE;
	gu8_OrionBMS2_Firmware_Patch			:BYTE;
	gu8_OrionBMS2_Constant_2				:BYTE;
	gu8_OrionBMS2_Constant_3				:BYTE;
	gu8_OrionBMS2_Constant_4				:BYTE;
	gu16_OrionBMS2_CheckSum					:UINT;
	gu8_OrionBMS2_Spare_6B6_7				:BYTE;
	// 6B9
	gu8_OrionBMS2_6B9_0: USINT;
	gu8_OrionBMS2_6B9_1: USINT;
	gu8_OrionBMS2_6B9_2: USINT;
	gu8_OrionBMS2_6B9_3: USINT;
	gu8_OrionBMS2_6B9_4: USINT;
	gu8_OrionBMS2_6B9_5: USINT;
	gu8_OrionBMS2_6B9_6: USINT;
	gu8_OrionBMS2_6B9_7: USINT;
	// 6BA
	gu8_OrionBMS2_6BA_0: USINT;
	gu8_OrionBMS2_6BA_1: USINT;
	gu8_OrionBMS2_6BA_2: USINT;
	gu8_OrionBMS2_6BA_3: USINT;
	gu8_OrionBMS2_6BA_4: USINT;
	gu8_OrionBMS2_6BA_5: USINT;
	gu8_OrionBMS2_6BA_6: USINT;
	gu8_OrionBMS2_6BA_7: USINT;
	// 6BB
	gu8_OrionBMS2_6BB_0: USINT;
	gu8_OrionBMS2_6BB_1: USINT;
	gu8_OrionBMS2_6BB_2: USINT;
	gu8_OrionBMS2_6BB_3: USINT;
	gu8_OrionBMS2_6BB_4: USINT;
	gu8_OrionBMS2_6BB_5: USINT;
	gu8_OrionBMS2_6BB_6: USINT;
	gu8_OrionBMS2_6BB_7: USINT;
	// 6BC
	gu8_OrionBMS2_6BC_0: USINT;
	gu8_OrionBMS2_6BC_1: USINT;
	gu8_OrionBMS2_6BC_2: USINT;
	gu8_OrionBMS2_6BC_3: USINT;
	gu8_OrionBMS2_6BC_4: USINT;
	gu8_OrionBMS2_6BC_5: USINT;
	gu8_OrionBMS2_6BC_6: USINT;
	gu8_OrionBMS2_6BC_7: USINT;
	// 6BD
	gu8_OrionBMS2_6BD_0: USINT;
	gu8_OrionBMS2_6BD_1: USINT;
	gu8_OrionBMS2_6BD_2: USINT;
	gu8_OrionBMS2_6BD_3: USINT;
	gu8_OrionBMS2_6BD_4: USINT;
	gu8_OrionBMS2_6BD_5: USINT;
	gu8_OrionBMS2_6BD_6: USINT;
	gu8_OrionBMS2_6BD_7: USINT;
	
	
	
	
	(**********************************************************)
	(*Rx Conversion*)
	gr_OrionBMS2_PackVoltage			:	REAL;
	gr_OrionBMS2_PackCurrent			:	REAL;
	gr_OrionBMS2_PackSOC				:	REAL;
	gr_OrionBMS2_Max_Charging_Voltage	:	REAL;
	
	(*DTC1 Flags*)
	OrionBMS2_DTCFlag1_0A07_DischargeLimitEnforcementFault1		:	BOOL;
	OrionBMS2_DTCFlag1_0A08_ChargerSafetyRelayFault1 			:	BOOL;
	OrionBMS2_DTCFlag1_0A09_InternalHardwareFault1				:	BOOL;
	OrionBMS2_DTCFlag1_0A0A_InternalHeatskinkThermistorFault 	:	BOOL;
	OrionBMS2_DTCFlag1_0A0B_InternalSoftwareFault1				:	BOOL;
	OrionBMS2_DTCFlag1_0A0C_HighestCellVoltageTooHighFault1 	:	BOOL;
	OrionBMS2_DTCFlag1_0A0E_LowestCellVoltageTooLowFault 		:	BOOL;
	OrionBMS2_DTCFlag1_0A10_PackTooHotFault1 					:	BOOL;
	OrionBMS2_DTCFlags_Reserved_Bit8 							:	BOOL;
	OrionBMS2_DTCFlags_Reserved_Bit9 							:	BOOL;
	OrionBMS2_DTCFlags_Reserved_Bit10 							:	BOOL;
	OrionBMS2_DTCFlags_Reserved_Bit11 							:	BOOL;
	OrionBMS2_DTCFlags_Reserved_Bit12 							:	BOOL;
	OrionBMS2_DTCFlags_Reserved_Bit13 							:	BOOL;
	OrionBMS2_DTCFlags_Reserved_Bit14 							:	BOOL;
	OrionBMS2_DTCFlags_Reserved_Bit15							:	BOOL;
	(*DTC2 Flags*)
	OrionBMS2_DTCFlags2_0A1F_InternalCommunicationFault			:	BOOL;
	OrionBMS2_DTCFlags2_0A12_CellBalancingStruckOffFault		:	BOOL;
	OrionBMS2_DTCFlags2_0A80_WeakCellFault						:	BOOL;
	OrionBMS2_DTCFlags2_0AFA_LowCellVoltageFault				:	BOOL;
	OrionBMS2_DTCFlags2_0A04_OpenWiringFault					:	BOOL;
	OrionBMS2_DTCFlags2_0AC0_CurrentSensorFault					:	BOOL;
	OrionBMS2_DTCFlags2_0A0D_HighestCellVoltageOver5vFault		:	BOOL;
	OrionBMS2_DTCFlags2_0A0F_CellASICFault						:	BOOL;
	OrionBMS2_DTCFlags2_0A02_WeakPackFault						:	BOOL;
	OrionBMS2_DTCFlags2_0A81_FanMonitorFault					:	BOOL;
	OrionBMS2_DTCFlags2_0A9C_ThermistorFault					:	BOOL;
	OrionBMS2_DTCFlags2_0100_ExternalCommunicationFault			:	BOOL;
	OrionBMS2_DTCFlags2_0560_RedundantPowerSupplyFault			:	BOOL;
	OrionBMS2_DTCFlags2_0AA6_HighVoltageIsolatonFault			:	BOOL;
	OrionBMS2_DTCFlags2_0A05_InputPowerSupplyFault				:	BOOL;
	OrionBMS2_DTCFlags2_0A06_ChargeLimitEnforcementFault		:	BOOL;
	
	(**********************************************************************)
	
	(* Current Limit Status *)
	gq_BMS2_BalActive			:BOOL;
	gq_BMS2_Flag_1				:BOOL;
	gq_BMS2_Flag_2				:BOOL;
	gq_BMS2_Flag_3				:BOOL;
	gq_BMS2_Flag_4				:BOOL;
	gq_BMS2_Flag_5				:BOOL;
	gq_BMS2_Flag_6				:BOOL;
	gq_BMS2_Flag_7				:BOOL;
	
	(********************************************************************)
	
	gq_OrionBMS2_CommsLoss										:	BOOL;
	// Tx
	gu8_BMS2_MPO_1_State					: USINT;
	// Tx
	gu8_BMS2_MPO_2_State					: USINT;
	// Tx
	gu8_BMS2_MPO_3_State					: USINT;
	// Tx
	gu8_BMS2_MPO_4_State					: USINT;
	// Tx
	gu8_BMS2_MPE_State					: USINT;
END_VAR

// Application/UserCode/BMS/CATL/CATLBMS_VAR_1
{attribute 'qualified_only'}
VAR_GLOBAL
END_VAR

// Application/UserCode/BMS/OrionBMS/OrionBMS1_VAR_1
VAR_GLOBAL
	(*Orion BMS1 Variables*)
	(******************************************)
	(*Rx*)
	(*6B0*)
	gs16_OrionBMS1_PackCurrent	:	INT;
	gu16_OrionBMS1_RAW_Pack_Voltage	:	UINT;
	gu8_OrionBMS1_RAW_SOC	:	USINT;
	gu16_OrionBMS1_RelayState	:	UINT;
	gu8_OrionBMS1_Custom_Flag_1	:	USINT;
	(*6B1*)
	gu8_OrionBMS1_Isolation_ADC			:	UINT;
	gu8_OrionBMS1_Shortest_Wave			:	UINT;
	gu16_OrionBMS1_Isolation_Clipping	:	UINT;
	gu16_OrionBMS1_Isolation_Threshold 	: UINT;
	(*6B2*)
	gu16_OrionBMS1_DTC_Flags1			:	UINT;
	gu16_OrionBMS1_DTC_Flags2			:	UINT;
	gu16_OrionBMS1_FailsafeStatus		:	UINT;
	gu16_OrionBMS1_Current_Limit_Status	:	UINT;
	(*6B3*)
	gu8_OrionBMS1_PackHealth			:	USINT;
	gu16_OrionBMS1_PackCycles			:	UINT;
	gu16_OrionBMS1_PackResistance		:	UINT;
	gu8_OrionBMS1_PopulatedCells		:	USINT;
	gu16_OrionBMS1_MaximumPackVoltage	:	UINT;
	(*6B4*)
	gu8_OrionBMS1_HighTemp				:	USINT;
	gu8_OrionBMS1_LowTemp				:	USINT;
	gu8_OrionBMS1_AverageTemp			:	USINT;
	gu8_OrionBMS1_InternalTemp			:	USINT;
	gu16_OrionBMS1_MinimumPackVoltage	:	UINT;  (*minimumPackvoltage*)
	gu16_OrionBMS1_PackAmphours			:	UINT;
	(*6B5*)
	gu16_OrionBMS1_AverageCellVoltage	:	UINT;
	gu16_OrionBMS1_LowCellVoltage		:	UINT;
	gu16_OrionBMS1_HighCellVoltage		:	UINT;
	gu8_OrionBMS1_LowCellVoltNumber		:	USINT;
	gu8_OrionBMS1_HighCellVoltNumber	:	USINT;
	(*6B6*)
	gu8_OrionBMS1_Low_Intres_ID				:	BYTE;
	gu8_OrionBMS1_High_Intres_ID			:	BYTE;
	gu16_OrionBMS1_Low_Cell_Resistance		:	UINT;
	gu16_OrionBMS1_High_Cell_Resistance		:	UINT;
	gu16_OrionBMS1_Average_Cell_Resistance	: 	UINT;
	
	(*6B7*)
	gu8_OrionBMS1_Low_Thermistor_ID			:	BYTE;
	gu8_OrionBMS1_High_Thermistor_ID		:	BYTE;
	gu16_OrionBMS1_PackDCL					:	UINT;
	gu16_OrionBMS1_PackCCL					:	UINT;
	gu16_OrionBMS1_PackSummedVoltage		:	UINT;
	// Constant will need checking after I am dead
	gu8_OrionBMS1_Firmware_Major: BYTE := 3;
	
	(*6B8*)
	gu8_OrionBMS1_Firmware_Minor			:BYTE;
	gu8_OrionBMS1_Firmware_Patch			:BYTE;
	gu8_OrionBMS1_Constant_2				:BYTE;// This is profile version will need manually inputting on BMS SW.
	gu8_OrionBMS1_Constant_3				:BYTE;// This is profile version will need manually inputting on BMS SW.
	gu8_OrionBMS1_Constant_4				:BYTE;// This is profile version will need manually inputting on BMS SW.
	gu16_OrionBMS1_CheckSum		:UINT;
	// Not USED Spare
	gu8_OrionBMS1_Spare_6B6_7				:BYTE;
	// 6B9 Not USED Spare
	gu8_OrionBMS1_6B9_0: USINT;
	// Not USED Spare
	gu8_OrionBMS1_6B9_1: USINT;
	// Not USED Spare
	gu8_OrionBMS1_6B9_2: USINT;
	gu8_OrionBMS1_6B9_3: USINT;
	gu8_OrionBMS1_6B9_4: USINT;
	// Not USED Spare
	gu8_OrionBMS1_6B9_5: USINT;
	gu8_OrionBMS1_6B9_6: USINT;
	gu8_OrionBMS1_6B9_7: USINT;
	// 6BA Not USED Spare
	gu8_OrionBMS1_6BA_0: USINT;
	gu8_OrionBMS1_6BA_1: USINT;
	gu8_OrionBMS1_6BA_2: USINT;
	gu8_OrionBMS1_6BA_3: USINT;
	gu8_OrionBMS1_6BA_4: USINT;
	// Not USED Spare
	gu8_OrionBMS1_6BA_5: USINT;
	gu8_OrionBMS1_6BA_6: USINT;
	gu8_OrionBMS1_6BA_7: USINT;
	// 6BB Not USED Spare
	gu8_OrionBMS1_6BB_0: USINT;
	gu8_OrionBMS1_6BB_1: USINT;
	gu8_OrionBMS1_6BB_2: USINT;
	gu8_OrionBMS1_6BB_3: USINT;
	gu8_OrionBMS1_6BB_4: USINT;
	gu8_OrionBMS1_6BB_5: USINT;
	gu8_OrionBMS1_6BB_6: USINT;
	gu8_OrionBMS1_6BB_7: USINT;
	// 6BC Not USED Spare
	gu8_OrionBMS1_6BC_0: USINT;
	gu8_OrionBMS1_6BC_1: USINT;
	gu8_OrionBMS1_6BC_2: USINT;
	gu8_OrionBMS1_6BC_3: USINT;
	gu8_OrionBMS1_6BC_4: USINT;
	gu8_OrionBMS1_6BC_5: USINT;
	gu8_OrionBMS1_6BC_6: USINT;
	gu8_OrionBMS1_6BC_7: USINT;
	// 6BD Not USED Spare
	gu8_OrionBMS1_6BD_0: USINT;
	gu8_OrionBMS1_6BD_1: USINT;
	gu8_OrionBMS1_6BD_2: USINT;
	gu8_OrionBMS1_6BD_3: USINT;
	gu8_OrionBMS1_6BD_4: USINT;
	gu8_OrionBMS1_6BD_5: USINT;
	gu8_OrionBMS1_6BD_6: USINT;
	gu8_OrionBMS1_6BD_7: USINT;
	
	
	
	(**********************************************************)
	(*Rx Conversion*)
	
	
	(*DTC1 Flags*)
	OrionBMS1_DTCFlag1_0A07_DischargeLimitEnforcementFault		:	BOOL;
	OrionBMS1_DTCFlag1_0A08_ChargerSafetyRelayFault 			:	BOOL;
	OrionBMS1_DTCFlag1_0A09_InternalHardwareFault				:	BOOL;
	OrionBMS1_DTCFlag1_0A0A_InternalHeatskinkThermistorFault 	:	BOOL;
	OrionBMS1_DTCFlag1_0A0B_InternalSoftwareFault				:	BOOL;
	OrionBMS1_DTCFlag1_0A0C_HighestCellVoltageTooHighFault 	:	BOOL;
	OrionBMS1_DTCFlag1_0A0E_LowestCellVoltageTooLowFault 		:	BOOL;
	OrionBMS1_DTCFlag1_0A10_PackTooHotFault 					:	BOOL;
	OrionBMS1_DTCFlags_Reserved_Bit8 							:	BOOL;
	OrionBMS1_DTCFlags_Reserved_Bit9 							:	BOOL;
	OrionBMS1_DTCFlags_Reserved_Bit10 							:	BOOL;
	OrionBMS1_DTCFlags_Reserved_Bit11 							:	BOOL;
	OrionBMS1_DTCFlags_Reserved_Bit12 							:	BOOL;
	OrionBMS1_DTCFlags_Reserved_Bit13 							:	BOOL;
	OrionBMS1_DTCFlags_Reserved_Bit14 							:	BOOL;
	OrionBMS1_DTCFlags_Reserved_Bit15							:	BOOL;
	(*DTC2 Flags*)
	OrionBMS1_DTCFlags2_0A1F_InternalCommunicationFault			:	BOOL;
	OrionBMS1_DTCFlags2_0A12_CellBalancingStruckOffFault		:	BOOL;
	OrionBMS1_DTCFlags2_0A80_WeakCellFault						:	BOOL;
	OrionBMS1_DTCFlags2_0AFA_LowCellVoltageFault				:	BOOL;
	OrionBMS1_DTCFlags2_0A04_OpenWiringFault					:	BOOL;
	OrionBMS1_DTCFlags2_0AC0_CurrentSensorFault					:	BOOL;
	OrionBMS1_DTCFlags2_0A0D_HighestCellVoltageOver5vFault		:	BOOL;
	OrionBMS1_DTCFlags2_0A0F_CellASICFault						:	BOOL;
	OrionBMS1_DTCFlags2_0A02_WeakPackFault						:	BOOL;
	OrionBMS1_DTCFlags2_0A81_FanMonitorFault					:	BOOL;
	OrionBMS1_DTCFlags2_0A9C_ThermistorFault					:	BOOL;
	OrionBMS1_DTCFlags2_0100_ExternalCommunicationFault			:	BOOL;
	OrionBMS1_DTCFlags2_0560_RedundantPowerSupplyFault			:	BOOL;
	OrionBMS1_DTCFlags2_0AA6_HighVoltageIsolatonFault			:	BOOL;
	OrionBMS1_DTCFlags2_0A05_InputPowerSupplyFault				:	BOOL;
	OrionBMS1_DTCFlags2_0A06_ChargeLimitEnforcementFault		:	BOOL;
	
	(**********************************************************************)
	
	gq_OrionBMS1_CommsLoss										:	BOOL;
	
	// Tx
	gu8_BMS1_MPO_1_State					: USINT;
	// Not connected to Anything. But it's Here.
	gu8_BMS1_MPO_2_State					: USINT;
	// Tx
	gu8_BMS1_MPO_3_State					: USINT;
	// Tx
	gu8_BMS1_MPO_4_State					: USINT;
	// Tx
	gu8_BMS1_MPE_State					: USINT;
END_VAR

// Application/UserCode/BMS/OrionBMS/OrionBMS2_VAR_1
VAR_GLOBAL
	(*Orion BMS2 Variables*)
	(******************************************)
	(*Rx*)
	(*6B0*)
	gs16_OrionBMS2_PackCurrent	:	INT;
	gu16_OrionBMS2_PackVoltage	:	UINT;
	gu8_OrionBMS2_RAW_SOC	:	USINT;
	gu16_OrionBMS2_RelayState	:	UINT;
	gu8_OrionBMS2_Custom_Flag_1	:	USINT;
	(*6B1*)
	gu8_OrionBMS2_Isolation_ADC			:	UINT;
	gu8_OrionBMS2_Shortest_Wave			:	UINT;
	gu16_OrionBMS2_Isolation_Clipping	:	UINT;
	gu16_OrionBMS2_Isolation_Threshold 	: UINT;
	(*6B2*)
	gu16_OrionBMS2_DTC_Flags1		:	UINT;
	gu16_OrionBMS2_DTC_Flags2		:	UINT;
	gu16_OrionBMS2_FailsafeStatus	:	UINT;
	gu16_OrionBMS2_CurrentLimit		:	UINT;
	(*6B3*)
	gu8_OrionBMS2_PackHealth			:	USINT;
	gu16_OrionBMS2_PackCycles			:	UINT;
	gu16_OrionBMS2_PackResistance		:	UINT;
	gu8_OrionBMS2_PopulatedCells		:	USINT;
	gu16_OrionBMS2_MaximumPackVoltage	:	UINT;
	(*6B4*)
	gu8_OrionBMS2_HighTemp				:	USINT;
	gu8_OrionBMS2_LowTemp				:	USINT;
	gu8_OrionBMS2_AverageTemp			:	USINT;
	gu8_OrionBMS2_InternalTemp			:	USINT;
	gu16_OrionBMS2_MinimumPackVoltage	:	UINT;  (*minimumPackvoltage*)
	gu16_OrionBMS2_PackAmphours			:	UINT;
	(*6B5*)
	gu16_OrionBMS2_AverageCellVoltage	:	UINT;
	gu16_OrionBMS2_LowCellVoltage		:	UINT;
	gu16_OrionBMS2_HighCellVoltage		:	UINT;
	gu8_OrionBMS2_LowCellVoltNumber		:	USINT;
	gu8_OrionBMS2_HighCellVoltNumber	:	USINT;
	(*6B6*)
	gu8_OrionBMS2_Low_Intres_ID				:	BYTE;
	gu8_OrionBMS2_High_Intres_ID			:	BYTE;
	gu16_OrionBMS2_Low_Cell_Resistance		:	UINT;
	gu16_OrionBMS2_High_Cell_Resistance		:	UINT;
	gu16_OrionBMS2_Average_Cell_Resistance	: 	UINT;
	
	(*6B7*)
	gu8_OrionBMS2_Low_Thermistor_ID			:	BYTE;
	gu8_OrionBMS2_High_Thermistor_ID		:	BYTE;
	gu16_OrionBMS2_PackDCL					:	UINT;
	gu16_OrionBMS2_PackCCL					:	UINT;
	gu16_OrionBMS2_PackSummedVoltage		:	UINT;
	
	(*6B8*)
	gu8_OrionBMS2_Firmware_Minor			:BYTE;
	gu8_OrionBMS2_Firmware_Patch			:BYTE;
	gu8_OrionBMS2_Constant_2				:BYTE;
	gu8_OrionBMS2_Constant_3				:BYTE;
	gu8_OrionBMS2_Constant_4				:BYTE;
	gu16_OrionBMS2_CheckSum					:UINT;
	gu8_OrionBMS2_Spare_6B6_7				:BYTE;
	// 6B9
	gu8_OrionBMS2_6B9_0: USINT;
	gu8_OrionBMS2_6B9_1: USINT;
	gu8_OrionBMS2_6B9_2: USINT;
	gu8_OrionBMS2_6B9_3: USINT;
	gu8_OrionBMS2_6B9_4: USINT;
	gu8_OrionBMS2_6B9_5: USINT;
	gu8_OrionBMS2_6B9_6: USINT;
	gu8_OrionBMS2_6B9_7: USINT;
	// 6BA
	gu8_OrionBMS2_6BA_0: USINT;
	gu8_OrionBMS2_6BA_1: USINT;
	gu8_OrionBMS2_6BA_2: USINT;
	gu8_OrionBMS2_6BA_3: USINT;
	gu8_OrionBMS2_6BA_4: USINT;
	gu8_OrionBMS2_6BA_5: USINT;
	gu8_OrionBMS2_6BA_6: USINT;
	gu8_OrionBMS2_6BA_7: USINT;
	// 6BB
	gu8_OrionBMS2_6BB_0: USINT;
	gu8_OrionBMS2_6BB_1: USINT;
	gu8_OrionBMS2_6BB_2: USINT;
	gu8_OrionBMS2_6BB_3: USINT;
	gu8_OrionBMS2_6BB_4: USINT;
	gu8_OrionBMS2_6BB_5: USINT;
	gu8_OrionBMS2_6BB_6: USINT;
	gu8_OrionBMS2_6BB_7: USINT;
	// 6BC
	gu8_OrionBMS2_6BC_0: USINT;
	gu8_OrionBMS2_6BC_1: USINT;
	gu8_OrionBMS2_6BC_2: USINT;
	gu8_OrionBMS2_6BC_3: USINT;
	gu8_OrionBMS2_6BC_4: USINT;
	gu8_OrionBMS2_6BC_5: USINT;
	gu8_OrionBMS2_6BC_6: USINT;
	gu8_OrionBMS2_6BC_7: USINT;
	// 6BD
	gu8_OrionBMS2_6BD_0: USINT;
	gu8_OrionBMS2_6BD_1: USINT;
	gu8_OrionBMS2_6BD_2: USINT;
	gu8_OrionBMS2_6BD_3: USINT;
	gu8_OrionBMS2_6BD_4: USINT;
	gu8_OrionBMS2_6BD_5: USINT;
	gu8_OrionBMS2_6BD_6: USINT;
	gu8_OrionBMS2_6BD_7: USINT;
	
	
	
	
	(**********************************************************)
	(*Rx Conversion*)
	
	(*DTC1 Flags*)
	OrionBMS2_DTCFlag1_0A07_DischargeLimitEnforcementFault		:	BOOL;
	OrionBMS2_DTCFlag1_0A08_ChargerSafetyRelayFault 			:	BOOL;
	OrionBMS2_DTCFlag1_0A09_InternalHardwareFault				:	BOOL;
	OrionBMS2_DTCFlag1_0A0A_InternalHeatskinkThermistorFault 	:	BOOL;
	OrionBMS2_DTCFlag1_0A0B_InternalSoftwareFault				:	BOOL;
	OrionBMS2_DTCFlag1_0A0C_HighestCellVoltageTooHighFault 	:	BOOL;
	OrionBMS2_DTCFlag1_0A0E_LowestCellVoltageTooLowFault 		:	BOOL;
	OrionBMS2_DTCFlag1_0A10_PackTooHotFault 					:	BOOL;
	OrionBMS2_DTCFlags_Reserved_Bit8 							:	BOOL;
	OrionBMS2_DTCFlags_Reserved_Bit9 							:	BOOL;
	OrionBMS2_DTCFlags_Reserved_Bit10 							:	BOOL;
	OrionBMS2_DTCFlags_Reserved_Bit11 							:	BOOL;
	OrionBMS2_DTCFlags_Reserved_Bit12 							:	BOOL;
	OrionBMS2_DTCFlags_Reserved_Bit13 							:	BOOL;
	OrionBMS2_DTCFlags_Reserved_Bit14 							:	BOOL;
	OrionBMS2_DTCFlags_Reserved_Bit15							:	BOOL;
	(*DTC2 Flags*)
	OrionBMS2_DTCFlags2_0A1F_InternalCommunicationFault			:	BOOL;
	OrionBMS2_DTCFlags2_0A12_CellBalancingStruckOffFault		:	BOOL;
	OrionBMS2_DTCFlags2_0A80_WeakCellFault						:	BOOL;
	OrionBMS2_DTCFlags2_0AFA_LowCellVoltageFault				:	BOOL;
	OrionBMS2_DTCFlags2_0A04_OpenWiringFault					:	BOOL;
	OrionBMS2_DTCFlags2_0AC0_CurrentSensorFault					:	BOOL;
	OrionBMS2_DTCFlags2_0A0D_HighestCellVoltageOver5vFault		:	BOOL;
	OrionBMS2_DTCFlags2_0A0F_CellASICFault						:	BOOL;
	OrionBMS2_DTCFlags2_0A02_WeakPackFault						:	BOOL;
	OrionBMS2_DTCFlags2_0A81_FanMonitorFault					:	BOOL;
	OrionBMS2_DTCFlags2_0A9C_ThermistorFault					:	BOOL;
	OrionBMS2_DTCFlags2_0100_ExternalCommunicationFault			:	BOOL;
	OrionBMS2_DTCFlags2_0560_RedundantPowerSupplyFault			:	BOOL;
	OrionBMS2_DTCFlags2_0AA6_HighVoltageIsolatonFault			:	BOOL;
	OrionBMS2_DTCFlags2_0A05_InputPowerSupplyFault				:	BOOL;
	OrionBMS2_DTCFlags2_0A06_ChargeLimitEnforcementFault		:	BOOL;
	
	(**********************************************************************)
	
	gq_OrionBMS2_CommsLoss										:	BOOL;
	// Tx
	gu8_BMS2_MPO_1_State					: USINT;
	// Tx
	gu8_BMS2_MPO_2_State					: USINT;
	// Tx
	gu8_BMS2_MPO_3_State					: USINT;
	// Tx
	gu8_BMS2_MPO_4_State					: USINT;
	// Tx
	gu8_BMS2_MPE_State					: USINT;
END_VAR

// Application/UserCode/CAN4/Heater/Heater_VAR
VAR_GLOBAL
	gq_Heater_EnableBit	:	BOOL;
	gu8_Heater_Perc		:	USINT;
	gu8_Heater_Temp_Tx: USINT;
	gq_HeaterPumpEnable	:	BOOL;
END_VAR

// Application/UserCode/BELDCDC/BELDCDC_VAR
VAR_GLOBAL
	(*All the variables relating to the DCDC*)
	(********************************************)
	(*Rx*)
	(*FWS*)
	gq_BelDCDC_flt_InputUV			:	BOOL;
	gq_BelDCDC_flt_InputOV			:	BOOL;
	gq_BelDCDC_flt_OutputUV			:	BOOL;
	gq_BelDCDC_flt_OutputOV			:	BOOL;
	gq_BelDCDC_flt_OutputOC			:	BOOL;
	gq_BelDCDC_flt_OTP				:	BOOL;
	gq_BelDCDC_flt_I2CFault			:	BOOL;
	gq_BelDCDC_flt_CANFault			:	BOOL;
	gq_BelDCDC_flt_EEPROM_CRCFault	:	BOOL;
	gq_BelDCDC_flt_ShortCircuit		:	BOOL;
	gq_BelDCDC_flt_ThermistorFault	:	BOOL;
	gq_BelDCDC_flt_Overload			:	BOOL;
	gq_BelDCDC_flt_OutputOVLatch	:	BOOL;
	gq_BelDCDC_flt_ReversePolarity	:	BOOL;
	gq_BelDCDC_war_CoolantOTP		:	BOOL;
	gq_BelDCDC_war_CurrentLimiting	:	BOOL;
	gq_BelDCDC_sts_UnitEnabled		:	BOOL;
	gq_BelDCDC_sts_Wakeup			:	BOOL;
	gq_BelDCDC_sts_Fault			:	BOOL;
	gq_BelDCDC_sts_LatchedFault		:	BOOL;
	gq_BelDCDC_sts_RemoteShutdown	:	BOOL;
	gq_BelDCDC_sts_StartupInitDone	:	BOOL;
	gq_BelDCDC_sts_InputOK			:	BOOL;
	gq_BelDCDC_sts_HVILOK			:	BOOL;
	gq_BelDCDC_sts_ReversePolarity	:	BOOL;
	gq_BelDCDC_sts_Hiccup			:	BOOL;
	(*IO*)
	gu16_BelDCDC_OutputVoltage_Rx	:	UINT;
	gu16_BelDCDC_OutputCurrent_Rx	:	UINT;
	gu16_BelDCDC_InputVoltage_Rx	:	UINT;
	gu16_BelDCDC_TempCoolant_Rx		:	UINT;
	(*Conversion*)
	gr_BelDCDC_OutputVoltage		:	REAL;
	gr_BelDCDC_OutputCurrent		:	REAL;
	gr_BelDCDC_InputVoltage			:	REAL;
	gr_BelDCDC_TempCoolant			:	REAL;
	
	gq_BELDCDC_CommsLoss			:	BOOL;
END_VAR

// Application/UserCode/CAN1/CAN1_VAR
VAR_GLOBAL
	(*Tx variables*)
	(*EEC1*)
	gu8_ENG_EngineTorqueMode					:	USINT;
	gu8_ENG_ActlEngPrcntTorqueHghResolution_Tx	:	USINT;
	gu8_ENG_DriversDemandEnginePercentTorque	:	USINT;
	gu8_ENG_ActualEnginePercentTorque			:	USINT;
	gu16_ENG_EngineSpeed_Tx						:	UINT;
	gu8_ENG_SrcAddrOfCtrllingDevForEngCtrl		:	USINT;
	gu8_ENG_EngineStarterMode					:	USINT;
	gu8_ENG_EngineDemandPercentTorque			:	USINT;
	(*EEC2*)
	gu8_ENG_AccelPedal1LowIdleSwitch			:	USINT;
	gu8_ENG_AccelPedalKickdownSwitch			:	USINT;
	gu8_ENG_RoadSpeedLimitStatus				:	USINT;
	gu8_ENG_AccelPedal2LowIdleSwitch			:	USINT;
	gu8_ENG_AccelPedalPosition_Tx				:	USINT;
	gu8_ENG_EnginePercLoadCurrentSpeed			:	USINT;
	gu8_ENG_RemoteAccelPedalPosition_Tx			:	USINT;
	gu8_ENG_AccelPedalPosition2_Tx				:	USINT;
	gu8_ENG_VehicleAccelRateLimitStatus			:	USINT;
	gu8_ENG_MomentaryEngMaxPowEnableFeedback	:	USINT;
	gu8_ENG_DPFThermalManagementActive			:	USINT;
	gu8_ENG_SCRThermalManagementActive			:	USINT;
	gu8_ENG_ActualMaxAvailableEngPercTorque_Tx	:	USINT;
	gu8_ENG_EstimatedPumpingPercentTorque		:	USINT;
	(*EEC3*)
	gu8_ENG_NominalFrictionPercTorque				:	USINT;
	gu16_ENG_EngDesiredOperatingSpeed_Tx			:	UINT;
	gu8_ENG_EngDesiredOperatingSpeedAsymAdjust		:	USINT;
	gu8_ENG_EstEngParasiticLossPercTorque			:	USINT;
	gu16_ENG_Aftertreatment1ExhaustGasMassFlow_Tx	:	UINT;
	gu8_ENG_Aftertreatment1IntakeDewPoint			:	USINT;
	gu8_ENG_Aftertreatment1ExhaustDewPoint			:	USINT;
	gu8_ENG_Aftertreatment2IntakeDewPoint			:	USINT;
	gu8_ENG_Aftertreatment2ExhaustDewPoint			:	USINT;
	(*CCSS*)
	gu8_ENG_MaxVehicleSpeedLimit				:	USINT;
	gu8_ENG_CruiseControlHighSetSpeedLimit		:	USINT;
	gu8_ENG_CruiseControlLowSetSpeedLimit		:	USINT;
	
	(*Tx preconversion*)
	(*EEC1*)
	gr_ENG_ActlEngPrcntTorqueHghResolution		:	REAL;
	gr_ENG_EngineSpeed							:	REAL;
	(*EEC2*)
	gr_ENG_AccelPedalPosition1					:	REAL;
	gr_ENG_RemoteAccelPedalPosition				:	REAL;
	gr_ENG_AccelPedalPosition2					:	REAL;
	gr_ENG_ActualMaxAvailableEngPercTorque		:	REAL;
	(*EEC3*)
	gr_ENG_EngDesiredOperatingSpeed				:	REAL;
	gr_ENG_AfterTreatment1ExhaustGasMassFlow	:	REAL;
	
	
	(*Rx Variables*)
	gq_Dennis_Accel_NewData						:	BOOL;
	gu8_AccelPedal_Dennis_Rx					:	USINT;
	gq_BrakePedal_Dennis_Rx						:	BOOL;
	gu8_BrakePedal_Perc_Dennis_Rx				:	USINT;
	gu8_GearSelector_Dennis_Rx					:	USINT;
	gq_Neutral_Dennis_Rq						:	BOOL;
	gq_Drive_Dennis_Rq							:	BOOL;
	gq_Reverse_Dennis_Rq						:	BOOL;
	
	gu8_Dennis_AirPressureSusp_Rx				:	USINT;
	gu8_Dennis_AirPressureBrake1_Rx				:	USINT;
	gu8_Dennis_AirPressureBrake2_Rx				:	USINT;
	
	(*EBC1*)
	gu8_EBC1_ASREngineControlActive				:	USINT;
	gu8_EBC1_ASRBrakeControlActive				:	USINT;
	gu8_EBC1_ABSActive							:	USINT;
	gu8_EBC1_EBSBrakeSwitch						:	USINT;
	gu8_EBC1_BrakePedalPosition					:	USINT;
	gu8_EBC1_ABSOffroadSwitch					:	USINT;
	gu8_EBC1_ASROffroadSwitch					:	USINT;
	gu8_EBC1_ASRHillholderSwitch				:	USINT;
	gu8_EBC1_TractionControlOverrideSwtich		:	USINT;
	gu8_EBC1_AcceleratorInterlockSwitch			:	USINT;
	gu8_EBC1_EngineDerateSwitch					:	USINT;
	gu8_EBC1_EngineAuxiliaryShutdownSwitch		:	USINT;
	gu8_EBC1_RemoteAcceleratorEnableSwitch		:	USINT;
	gu8_EBC1_EngineRetarderSelection			:	USINT;
	gu8_EBC1_ABSFullyOperational				:	USINT;
	gu8_EBC1_gu8_EBC1_EBSRedWarningSignal		:	USINT;
	gu8_EBC1_ABSEBSAmberWarningSignal			:	USINT;
	gu8_EBC1_ATCASRInformationSignal			:	USINT;
	gu8_EBC1_SrcAddrOfCrtllingDevForBrkCtrl		:	USINT;
	gu8_EBC1_HaltBrakeSwitch					:	USINT;
	gu8_EBC1_TrailerABSStatus					:	USINT;
	gu8_EBC1_TractorMntdTrailerABSWarningSignal	:	USINT;
	
	(*EBC2*)
	gu16_EBC2_KB_FrontAxleSpeed_Rx				:	UINT;
	gu16_EBC2_KB_FrontLeftRelSpd_Rx				:	USINT;
	gu16_EBC2_KB_FrontRightRelSpd_Rx			:	USINT;
	gu16_EBC2_KB_RearLeft1RelSpd_Rx				:	USINT;
	gu16_EBC2_KB_RearRight1RelSpd_Rx			:	USINT;
	gu16_EBC2_KB_RearLeft2RelSpd_Rx				:	USINT;
	gu16_EBC2_KB_RearRight2RelSpd_Rx			:	USINT;
	
	gr_EBC2_KB_FrontAxleSpeed				:	REAL;
	gr_EBC2_KB_FrontLeftRelSpd				:	REAL;
	gr_EBC2_KB_FrontRightRelSpd				:	REAL;
	gr_EBC2_KB_RearLeft1RelSpd				:	REAL;
	gr_EBC2_KB_RearRight1RelSpd				:	REAL;
	gr_EBC2_KB_RearLeft2RelSpd				:	REAL;
	gr_EBC2_KB_RearRight2RelSpd				:	REAL;
	
	gu8_RegenStick01Pos						:	USINT;
	gu8_RegenStick12Pos						:	USINT;
	
	(*Dennis CAN1 Comms loss*)
	gq_Dennis_CAN1_CommsLoss					:	BOOL;
	
	gq_ABSActive								:	BOOL;
	
	(*Allison*)
	gu8_ETC7_TransmissionEngaged_Tx				:	USINT;
	gu8_ProbA_GearSelected_Tx					:	USINT;

	
	gq_Bob_Handbrake_CAN	:	BOOL;
	gq_Bob_Brake_CAN		:	BOOL;
	gu8_Bob_BrakePos_CAN	:	USINT;
	
	gu8_Bob_Accel_CAN		:	USINT;
	gr_Bob_Accel			:	REAL;
	gu8_Bob_RegenSelector_CAN	:	USINT;
	
	gu16_Bob_RightDrive_CAN	:	UINT;
	gu16_Bob_LeftDrive_CAN	:	UINT;
	gu16_Bob_RightFront_CAN	:	UINT;
	gu16_Bob_LeftFront_CAN	:	UINT;
	
	gu8_Bob_ServiceBrakeAirPressCircuit1_CAN	:	USINT;
	gu8_Bob_ServiceBrakeAirPressCircuit2_CAN	:	USINT;
	gu8_Bob_AirSuspensionSupplyPress_CAN		:	USINT;
	
	gr_Bob_ServiceBrakeAirPressCircuit1		:	REAL;
	gr_Bob_ServiceBrakeAirPressCircuit2		:	REAL;
	gr_Bob_AirSuspensionSupplyPress			:	REAL;
	
	gu8_Merc_AirComepressor_Rq	:	USINT;
	gq_Merc_AirComp_Rq		:	BOOL;
	gq_Merc_AirComp_Enabled	:	BOOL;
	
	gu16_RPM_Display	:	UINT;
	gq_StabTracDisable_Rx	:	BOOL;
	gq_Bob_WheelSpeedSensor_Fail	:	BOOL;
	
	gu16_MCM02_EngineTorque_Tx	:	UINT;
	gu16_TCM03_ShaftSpeed_Tx	:	UINT;
	
END_VAR

// Application/UserCode/CAN3/CAN3_VAR
VAR_GLOBAL
	
	gu8_GearSelector_Bob_Rx	:	USINT	:=	0;
	gq_Neutral_Bob_Rq	:	BOOL;
	gq_Drive_Bob_Rq		:	BOOL;
	gq_Reverse_Bob_Rq	:	BOOL;
	
	gu8_Merc_AutoManualSwitch	:	USINT;
	gu8_Merc_GearSelectSwitch	:	USINT;
	gq_Merc_Neutral				:	BOOL;
	gq_Merc_Drive				:	BOOL;
	gq_Merc_Reverse				:	BOOL;
END_VAR

// Application/UserCode/Main Program/Main_VAR
VAR_GLOBAL
	gu8_SystemState	:	USINT	:=	0;
	gq_SystemError	:	BOOL	:=	FALSE;
	gq_ParkBrake	:	BOOL;
	
	gr_VehicleSpeed_kmph	:	REAL;
	
	(*Chassis Paramters*)
	gq_HandBrake			:	BOOL	:=	FALSE;
	gq_BrakeSwitch			:	BOOL	:=	FALSE;
	gu8_BrakePedal_Perc		:	USINT	:=	0;
	gr_AccelPedal_Perc		:	REAL	:=	0;
	
	gq_Gear_Drive_Rq		:	BOOL	:=	FALSE;
	gq_Gear_Reverse_Rq		:	BOOL	:=	FALSE;
	gq_Gear_Neutral_Rq		:	BOOL	:=	FALSE;
	
	gr_J1939_AirSuspensionSupplyPress		:	REAL;
	gr_J1939_ServiceBrakeAirPressCircuit1	:	REAL;
	gr_J1939_ServiceBrakeAirPressCircuit2	:	REAL;
	gq_Bob_AirCompressorStatus_CAN			:	BOOL;
	
	gu8_RegenSelector		:	USINT;
	
	gs16_MaxTemp_degC		:	INT;
	
	gr_LowAirPressure_Intro		: REAL;
	gr_HighAirPressure_CutOff	: REAL;
	
	gq_EStop			:	BOOL;
	gq_EStopLatch		:	BOOL;
	gq_BodySteps		:	BOOL;
	gq_ReverseLights	:	BOOL;
	
	(*Contactor Return*)
	gq_BMS1_AuxPosContactor		:	BOOL;
	gq_BMS1_AuxNegContactor		:	BOOL;
	gq_BMS2_AuxPosContactor		:	BOOL;
	gq_BMS2_AuxNegContactor		:	BOOL;
	
END_VAR
VAR_GLOBAL CONSTANT
	STANDBY_SYS		:	USINT	:=	0;
	DRIVE_SYS		:	USINT	:=	1;
	PLUGIN_SYS		:	USINT	:=	2;
	ERROR_SYS		:	USINT	:=	3;
	OFF_SYS			:	USINT	:=	4;
	
	BMS_ORION		:	USINT	:=	1;
	BMS_ACTIA		:	USINT	:=	2;
	
	CHASSIS_DENNIS	:	USINT	:=	1;
	CHASSIS_BOB		:	USINT	:=	2;
	CHASSIS_IVECO	:	USINT	:=	4;
	CHASSIS_DAF		:	USINT	:=	8;
	CHASSIS_ISUZU	:	USINT	:=	16;
	CHASSIS_ESTARGLIDER : USINT :=	32;
	
	CHARGER_BRUSA	:	USINT	:=	1;
END_VAR

// Application/UserCode/MCU/MCU_VAR
VAR_GLOBAL
	(********************************************************)
	(*Rx*)
	(*MCUCommandResponse*)
	gu8_MCU_State						:	USINT;
	gu8_MCU_OperationalMode				:	USINT;
	gq_MCU_RegenDeratingStatus			:	BOOL;
	gu8_MCU_RegenDerating				:	USINT;
	gu8_MCU_TractionDerating			:	USINT;
	gu16_MCU_MaxMotorSpeedForward_Rx	:	UINT;
	gu16_MCU_MaxMotorSpeedReverse_Rx	:	UINT;
	gq_MCU_MaxMotorSpeedForwardStatus	:	BOOL;
	gq_MCU_MaxMotorSpeedReverseStatus	:	BOOL;
	gq_MCU_TractionDeratingStatus		:	BOOL;
	gu8_MCU_RollingCounter_Comm1		:	USINT;
	(*MCUCommandResponse2*)
	gu16_MCU_MotorSpeed_Rx				:	UINT;
	gu16_MCU_MotorAngle_Rx				:	UINT;
	gq_MVU_MotorAngleStatus				:	BOOL;
	gq_MCU_MotorSpeedStatus				:	BOOL;
	gq_MCU_SpeedReductionRequest		:	BOOL;
	gq_MCU_EmergencyStop				:	BOOL;
	gu8_MCU_RollingCounter_Comm2		:	USINT;
	(*MCUEventInfo1*)
	gq_MCU_Fault_PhaseToChassis					:	BOOL;
	gq_MCU_Fault_InterlockBatteryCable			:	BOOL;
	gq_MCU_Fault_InterlockMotorCable			:	BOOL;
	gq_MCU_Fault_DriveCoverWasOpened			:	BOOL;
	gq_MCU_Fault_PhaseToChassisStatus			:	BOOL;
	gq_MCU_Fault_InterlockBatteryCableStatus	:	BOOL;
	gq_MCU_Fault_InterlockMotorCableStatus		:	BOOL;
	gq_MCU_Fault_DriveCoverWasOpenedStatus		:	BOOL;
	(*MCUInfo1*)
	gu8_MCU_AuxiliaryVoltage_Rx					:	USINT;
	gu16_MCU_HighPowerVoltage					:	UINT;
	gq_MCU_HighPowerCurrentStatus				:	BOOL;
	gq_MCU_AuxiliaryVoltageStatus				:	BOOL;
	gq_MCU_HighPowerVoltageStatus				:	BOOL;
	gu16_MCU_HighPowerCurrent_Rx				:	UINT;
	gu8_MCU_RollingCounter_Info1				:	USINT;
	(*MCUInfo2*)
	gu16_MCU_MotorTorqueEstimated_Rx			:	UINT;
	gu16_MCU_TractionTorqueAvailable_Rx			:	UINT;
	gu16_MCU_RegenTorqueAvailable_Rx			:	UINT;
	gq_MCU_MotorTorqueEstimatedStatus			:	BOOL;
	gq_MCU_TractionTorqueAvailableStatus		:	BOOL;
	gq_MCU_RegenTorqueAvailableStatus			:	BOOL;
	gu8_MCU_RollingCounter_Info2				:	USINT;
	(*MCUOnEventInfo1*)
	gu16_MCU_EventID							:	UINT;
	gu8_MCU_RollingCounter_OnEventInfo1			:	USINT;
	(*MCUThermal1*)
	gu8_MCU_DriveCoolingFlowRequest_Rx			:	USINT;
	gu8_MCU_MotorCoolingFlowRequest_Rx			:	USINT;
	gu8_MCU_ThermalIndicator_Rx					:	USINT;
	gq_MCU_DriveCoolingFlowRequestStatus		:	BOOL;
	gq_MCU_MotorCoolingFlowRequestStatus		:	BOOL;
	gq_MCU_ThermalIndicatorStatus				:	BOOL;
	gu8_MCU_RollingCounter_Thermal1				:	USINT;
	(*MCUPollingMCUResponse*)
	gq_MCU_ResponseAcknowledgement				:	BOOL;
	gu8_MCU_MCUPollResponse_Multiplex			:	USINT;
		(*MCU MaxMotorSpeed*)
		gu16_MCU_MaxMotorSpeed_Rx				:	UINT;
		(*MCU MaxMotorTorque*)
		gu16_MCU_MaxMotorTorque_Rx				:	UINT;
		(*MCU ProtocolVersion*)
		gu8_MCU_MajorMCUProtocol				:	USINT;
		gu8_MCU_MinorMCUProtocol				:	USINT;
		gu8_MCU_ExtensionMajor					:	USINT;
		gu8_MCU_ExtensionMinor					:	USINT;
		(*MCU SWVersion1*)
		gu8_MCU_MajorMCUSW						:	USINT;
		gu8_MCU_MinorMCUSW						:	USINT;
		gu16_MCU_BranchMCUSW					:	UINT;
		(*MCU SWVersion2*)
		gu32_MCU_RevisionMCUSW					:	UDINT;
		(*MCU TotalMotorRotation*)
		gu32_MCU_TotalMotorRotation_LSB			:	UDINT;
		gu32_MCU_TotalMotorRotation_MSB			:	UDINT;
		gr_MCU_TotalMotorRotation_LSB			:	REAL;
		gr_MCU_TotalMotorRotation_MSB			:	REAL;
		gr_MCU_TotalMotorRotation				:	REAL;
		;
		(*MCUPollingVMU*)
		gu8_MCU_VMUBootNumber						:	USINT;
		(*VMUBootNumber*)
		gu16_MCU_BootNumber						:	UINT;
	
	(***************************************************************)
	(*Rx Conversion*)
	gr_MCU_MaxMotorSpeedForward		:	REAL;
	gr_MCU_MaxMotorSpeedReverse		:	REAL;
	gr_MCU_MotorSpeed				:	REAL;
	gr_MCU_MotorAngle				:	REAL;
	gr_MCU_AuxiliaryVoltage			:	REAL;
	gr_MCU_HighPowerCurrent			:	REAL;
	gr_MCU_MotorTorqueEstimated		:	REAL;
	gr_MCU_TractionTorqueAvailable	:	REAL;
	gr_MCU_RegenTorqueAvailable		:	REAL;
	gr_MCU_DriveCoolingFlowRequest	:	REAL;
	gr_MCU_MotorCoolingFlowRequest	:	REAL;
	gr_MCU_ThermalIndicator			:	REAL;
	gr_MCU_MaxMotorSpeed			:	REAL;
	gr_MCU_MaxMotorTorque			:	REAL;
	(****************************************************************)
	(*Tx*)
	(*VMU Comm1*)
	gu16_MCU_MaxChargeCurrent		:	UINT;
	gu8_MCU_OperationRequest		:	USINT;
	gu16_MCU_MaxDischargeCurrent	:	UINT;
	gu16_MCU_MaxBatteryVoltage		:	UINT;
	gq_MCU_MaxDiscahrgeCurrentStatus	:	BOOL;
	gq_MCU_MaxBatteryVoltageStatus	:	BOOL;
	gq_MCU_MinBatteryVoltageStatus	:	BOOL;
	gq_MCU_MaxChargeCurrentStatus	:	BOOL;
	gu16_MCU_MinBatteryVoltage		:	UINT;
	gu8_MCU_RollingCounter_VMUComm1	:	USINT;
	(*VMU Comm2*)
	gu8_MCU_OperationalMode_Tx		:	USINT;
	gu8_MCU_CommandMode				:	USINT;
	gq_MCU_SpeedCommandStatus		:	BOOL;
	gq_MCU_TorqueCommandStatus		:	BOOL;
	gu16_MCU_TorqueCommand_Tx		:	UINT;
	gu16_MCU_SpeedCommand_Tx		:	UINT;
	gu8_MCU_RollingCounter_VMUComm2	:	USINT;
	(*VMU CommandSafety*)
	gu16_MCU_ReferenceTorqueCommand_Tx	:	UINT;
	gu16_MCU_ReferenceSpeedCommand_Tx	:	UINT;
	gu8_MCU_ReferenceCommandMode		:	USINT;
	gu8_MCU_RollingCounter_VMUCommSafety	:	USINT;
	(*VMUPollingMCU*)
	gu8_MCU_VMUPollMCU_Multiplex	:	USINT;
		(*MCUMaxMotorSpeed*)
		gu16_MCU_MaxMotorSpeed_Tx	:	UINT;
		(*MCUMaxMotorTorque*)
		gu16_MCU_MaxMotorTorque_Tx	:	UINT;
		(*MCUProtocolVersion*)
		gu8_MCU_MajorMCUProtocol_Tx	:	USINT;
		gu8_MCU_MinorMCUProtocol_Tx	:	USINT;
		(*MCUSWVersion1*)
		gu8_MCU_MajorMCUSW_Tx			:	USINT;
		gu8_MCU_MinorMCUSW_Tx			:	USINT;
		gu16_MCU_BranchMCUSW_Tx			:	UINT;
		(*MCUSWVersion2*)
		gu32_MCU_RevisionMCUSW_Tx		:	UDINT;
		(*MCUTotalMotorRotation*)
		gu32_MCU_TotalMotorRotation_LSB_Tx	:	UDINT;
		gu32_MCU_TotalMotorRotation_MSB_Tx	:	UDINT;
	(*VMUPollingVMUResponse*)
	gq_MCU_PollVMUResponse_Acknowledgement	:	BOOL;
	gu8_MCU_PollVMUResponse_Multiplex		:	USINT;
		(*BootNumber*)
		gu16_MCU_BootNumber_Tx			:	UINT;		
	(*VMUSelectProtocolVersion*)
	gu8_MCU_SelectMajorMCUProtocol_Tx		:	USINT;
	gu8_MCU_SelectMinorMCUProtocol_Tx		:	USINT;
	
	(****************************************************************)
	(*True values - pre Tx*)
	gr_MCU_TorqueCommand_PreCF			:	REAL;
	gr_MCU_TorqueCommand_PreCF_Limited	:	REAL;
	gr_MCU_SpeedCommand_PreCF			:	REAL;
	gr_MCU_ReferenceTorqueCommand_PreCF	:	REAL;
	gr_MCU_ReferenceSpeedCommand_PreCF	:	REAL;
	gr_MCU_MaxMotorSpeed_PreCF			:	REAL;
	
	(****************************************************************)
	(*Latching Gear Selection*)
	gq_Gear_Neutral						:	BOOL;
	gq_Gear_Drive						:	BOOL;
	gq_Gear_DriveCrawl					:	BOOL;
	gq_Gear_Reverse						:	BOOL;
	gq_Gear_ReverseCrawl				:	BOOL;
	
	gq_MCU_CommsLoss					:	BOOL;
	
	(*Drivability*)
	gq_ABS_TorqueDisable				:	BOOL;
	
	gr_RearAxle_RelativeSpeed_kph		:	REAL;
	gu8_TractionLoss					:	USINT;
	gr_LeftWheels_RelativeSpeed_kph		:	REAL;
	gr_RightWheels_RelativeSpeed_kph	:	REAL;
	gu8_StabilityLoss					:	USINT;
	gq_ZeroTorqueRq						:	BOOL;
	gton_TorqueReIntro_Timer			:	TON;
	
	gr_RegenSOCMultiplier				:	REAL;
	gr_RegenMultiplierRq				:	REAL;
	gr_RegenIntroCF						:	REAL;
	gq_RegenActive						:	BOOL;
	gr_RegenSpeedDegrading				:	REAL;
	
	
	gr_VehicleTripDistance				:	REAL;
	gr_VehicleInitialTripDistance		:	REAL;
	
	gr_TorqueReIntro					:	REAL;
	gr_TorqueReIntroMax					:	REAL;
	
	gr_MCU_TorqueCommand_Limited	:	REAL;
	gr_MCU_PreviousTorqueCommand	:	REAL;
	
	gq_InitialProtocolGrab			:	BOOL;
END_VAR
VAR_GLOBAL CONSTANT
	MAXMOTORSPEED				:	USINT	:=	2;
	MAXMOTORTORQUE				:	USINT	:=	1;
	PROTOCOLVERSION				:	USINT	:=	0;
	SWVERSION1					:	USINT	:=	3;
	SWVERSION2					:	USINT	:=	4;
	TOTALMOTORROTATION			:	USINT	:=	5;
	TOTALMOTORROTATIONUSINTMCU	:	USINT	:=	6;
	
	VMUBOOTNUMBER				:	USINT	:=	0;
END_VAR

// Application/UserCode/Sevcon_PSP/Sevcon_Steer_VAR
VAR_GLOBAL
	(*********************************************************)
	
	(*Transmit*)
	(*Torque Demands 1*)
	gu16_Sevcon1_TorqueRq_Tx				:	UINT;
	gu16_Sevcon1_Controlword				:	UINT;
	gu16_Sevcon1_TorqueTractionLimit_Tx		:	UINT;
	gu8_Sevcon1_SEQCommand1					:	USINT;
	gu8_Sevcon1_CSCommand1					:	USINT;
	
	(*Torque Demands 2*)
	gu16_Sevcon1_TorqueRegenLimit_Tx		:	UINT;
	gu16_Sevcon1_SpeedLimitForward			:	UINT;
	gs16_Sevcon1_SpeedLimitReverse			:	INT;
	gu8_Sevcon1_SEQCommand2					:	USINT;
	gu8_Sevcon1_CSCommand2					:	USINT;
	
	(*Battery Demands*)
	gu16_Sevcon1_DCLink_ImaxDischarge		:	UINT;
	gs16_Sevcon1_DCLink_ImaxRecharge		:	INT;
	gu16_Sevcon1_DCLink_VoltageTarget_Tx	:	UINT;
	gu8_Sevcon1_SEQCurrentLimits			:	USINT;
	gu8_Sevcon1_CSCurrentLimits				:	USINT;
	
	(*I Demand Control*)
	gu16_Sevcon1_DebugIqDirectControl_Tx	:	UINT;
	gu16_Sevcon1_DebugIdDirectControl_Tx	:	UINT;
	gu8_Sevcon1_DirectCurrents				:	USINT;
	gu8_Sevcon1_CSDirectCurrents			:	USINT;
	
	(*********************************************************)
	
	(*Receive*)
	(*Torque Status 1*)
	gs16_Sevcon1_TorqueMeasured_Rx		:	INT;
	gs16_Sevcon1_SpeedMeasured			:	INT;
	gs16_Sevcon1_DCLink_Current			:	INT;
	gu8_Sevcon1_SEQ_Torque				:	USINT;
	gu8_Sevcon1_CS_Torque				:	USINT;
	
	(*Torque Status 2*)
	gs16_Sevcon1_TorqueAvailableForward_Rx	:	INT;
	gs16_Sevcon1_TorqueAvailableReverse_Rx	:	INT;
	gu8_Sevcon1_InverterStatus			:	USINT;
	gu8_Sevcon1_TorqueLimitCode			:	USINT;
	gu8_Sevcon1_SEQ_Status				:	USINT;
	gu8_Sevcon1_CS_Status				:	USINT;
	
	(*Temperature*)
	gs16_Sevcon1_TempRemaining			:	INT;
	gs16_Sevcon1_MotorTemp				:	INT;
	gs16_Sevcon1_DCLink_Voltage_Rx		:	INT;
	gu8_Sevcon1_SEQ_Temp					:	USINT;
	gu8_Sevcon1_CS_Temp					:	USINT;
	
	(**)
	gs16_Sevcon1_FaultCode				:	INT;
	gs32_Sevcon1_FaultData				:	DINT;
	gu8_Sevcon1_SEQ_Fault				:	USINT;
	gu8_Sevcon1_CS_Fault					:	USINT;
	
	(**)
	gs32_Sevcon1_EncoderPosition_Rx		:	DINT;
	
	(**)
	gs16_Sevcon1_Debug_Id_Act_Rx			:	INT;
	gs16_Sevcon1_Debug_Iq_Act_Rx			:	INT;
	gs16_Sevcon1_Debug_Id_Ref_Rx			:	INT;
	gs16_Sevcon1_Debug_Iq_Ref_Rx			:	INT;
	
	(**)
	gu8_Sevcon1_Debug_Temp_Junction0		:	USINT;
	gu8_Sevcon1_Debug_Temp_Junction1		:	USINT;
	gu8_Sevcon1_Debug_Temp_Junction2		:	USINT;
	gu8_Sevcon1_Debug_Temp_Junction3		:	USINT;
	gu8_Sevcon1_Debug_Temp_Junction4		:	USINT;
	gu8_Sevcon1_Debug_Temp_Junction5		:	USINT;
	gu8_Sevcon1_Debug_Temp_MotorMeasured	:	USINT;
	gu8_Sevcon1_Debug_Temp_MotorEstimate	:	USINT;
	
	(**)
	gu8_Sevcon1_Debug_Temp_CapEstimateFast	:	USINT;
	gu8_Sevcon1_Debug_Temp_Track				:	USINT;
	gu8_Sevcon1_Debug_Temp_CapEstimateSlow	:	USINT;
	gu8_Sevcon1_Debug_Temp_Heatsink			:	USINT;
	gu8_Sevcon1_Debug_Temp_DeltaTj			:	USINT;
	gu8_Sevcon1_Debug_Temp_Normalised		:	USINT;
	gu8_Sevcon1_Debug_Temp_Coolant			:	USINT;
	gu8_Sevcon1_Debug_Temp_Winding			:	USINT;
	
	(**)
	gs16_Sevcon1_Debug_MaxFlux				:	INT;
	gs16_Sevcon1_Debug_IvLim					:	INT;
	gs16_Sevcon1_Debug_IqMax					:	INT;
	gs16_Sevcon1_Debug_Ls_Rx					:	INT;
	
	(**)
	gs16_Sevcon1_Debug_Slip_Rx				:	INT;
	gs16_Sevcon1_Debug_LmSat_Rx				:	INT;
	gs16_Sevcon1_Debug_IqMax2				:	INT;
	gs16_Sevcon1_Debug_RecipFlux				:	INT;
	
	(*********************************************************)
	(*Tx conversion*)
	gr_Sevcon1_TorqueRq					:	REAL;
	gr_Sevcon1_TorqueTractionLimit		:	REAL;
	gr_Sevcon1_TorqueRegenLimit			:	REAL;
	gr_Sevcon1_DCLink_VoltageTarget		:	REAL;
	gr_Sevcon1_DebugIqDirectControl		:	REAL;
	gr_Sevcon1_DebugIdDirectControl		:	REAL;
	
	(*********************************************************)
	(*Rx converison*)
	gr_Sevcon1_TorqueMeasured			:	REAL;
	gr_Sevcon1_TorqueAvailableForward	:	REAL;
	gr_Sevcon1_TorqueAvailableReverse	:	REAL;
	gr_Sevcon1_DCLink_Voltage			:	REAL;
	gr_Sevcon1_EncoderPosition			:	REAL;
	gr_Sevcon1_Debug_Id_Act				:	REAL;
	gr_Sevcon1_Debug_Iq_Act				:	REAL;
	gr_Sevcon1_Debug_Id_Ref				:	REAL;
	gr_Sevcon1_Debug_Iq_Ref				:	REAL;
	gr_Sevcon1_Debug_Ls					:	REAL;
	gr_Sevcon1_Debug_Slip				:	REAL;
	gr_Sevcon1_Debug_LmSat				:	REAL;
	
	
	gq_Sevcon1_CommsLoss				:	BOOL;
	
END_VAR

// Application/UserCode/BMS/CATL/CATLBMS_VAR
{attribute 'qualified_only'}
VAR_GLOBAL
END_VAR

// Application/UserCode/BMS/OrionBMS/OrionBMS1_VAR
VAR_GLOBAL
	(*Orion BMS1 Variables*)
	(******************************************)
	(*Rx*)
	(*6B0*)
	gs16_OrionBMS1_PackCurrent	:	INT;
	gu16_OrionBMS1_RAW_Pack_Voltage	:	UINT;
	gu8_OrionBMS1_RAW_SOC	:	USINT;
	gu16_OrionBMS1_RelayState	:	UINT;
	gu8_OrionBMS1_Custom_Flag_1	:	USINT;
	(*6B1*)
	gu8_OrionBMS1_Isolation_ADC			:	UINT;
	gu8_OrionBMS1_Shortest_Wave			:	UINT;
	gu16_OrionBMS1_Isolation_Clipping	:	UINT;
	gu16_OrionBMS1_Isolation_Threshold 	: UINT;
	(*6B2*)
	gu16_OrionBMS1_DTC_Flags1			:	UINT;
	gu16_OrionBMS1_DTC_Flags2			:	UINT;
	gu16_OrionBMS1_FailsafeStatus		:	UINT;
	gu16_OrionBMS1_Current_Limit_Status	:	UINT;
	(*6B3*)
	gu8_OrionBMS1_PackHealth			:	USINT;
	gu16_OrionBMS1_PackCycles			:	UINT;
	gu16_OrionBMS1_PackResistance		:	UINT;
	gu8_OrionBMS1_PopulatedCells		:	USINT;
	gu16_OrionBMS1_MaximumPackVoltage	:	UINT;
	(*6B4*)
	gu8_OrionBMS1_HighTemp				:	USINT;
	gu8_OrionBMS1_LowTemp				:	USINT;
	gu8_OrionBMS1_AverageTemp			:	USINT;
	gu8_OrionBMS1_InternalTemp			:	USINT;
	gu16_OrionBMS1_MinimumPackVoltage	:	UINT;  (*minimumPackvoltage*)
	gu16_OrionBMS1_PackAmphours			:	UINT;
	(*6B5*)
	gu16_OrionBMS1_AverageCellVoltage	:	UINT;
	gu16_OrionBMS1_LowCellVoltage		:	UINT;
	gu16_OrionBMS1_HighCellVoltage		:	UINT;
	gu8_OrionBMS1_LowCellVoltNumber		:	USINT;
	gu8_OrionBMS1_HighCellVoltNumber	:	USINT;
	(*6B6*)
	gu8_OrionBMS1_Low_Intres_ID				:	BYTE;
	gu8_OrionBMS1_High_Intres_ID			:	BYTE;
	gu16_OrionBMS1_Low_Cell_Resistance		:	UINT;
	gu16_OrionBMS1_High_Cell_Resistance		:	UINT;
	gu16_OrionBMS1_Average_Cell_Resistance	: 	UINT;
	
	(*6B7*)
	gu8_OrionBMS1_Low_Thermistor_ID			:	BYTE;
	gu8_OrionBMS1_High_Thermistor_ID		:	BYTE;
	gu16_OrionBMS1_PackDCL					:	UINT;
	gu16_OrionBMS1_PackCCL					:	UINT;
	gu16_OrionBMS1_PackSummedVoltage		:	UINT;
	// Constant will need checking after I am dead
	gu8_OrionBMS1_Firmware_Major: BYTE := 3;
	
	(*6B8*)
	gu8_OrionBMS1_Firmware_Minor			:BYTE;
	gu8_OrionBMS1_Firmware_Patch			:BYTE;
	// This is profile version will need manually inputting on BMS SW.
	gu8_OrionBMS1_Constant_2				:BYTE := 7;
	// This is profile version will need manually inputting on BMS SW.
	gu8_OrionBMS1_Constant_3				:BYTE := 0;
	// This is profile version will need manually inputting on BMS SW.
	gu8_OrionBMS1_Constant_4				:BYTE := 0;
	gu16_OrionBMS1_CheckSum		:UINT;
	// Not USED Spare
	gu8_OrionBMS1_Spare_6B6_7				:BYTE;
	// 6B9 Not USED Spare
	gu8_OrionBMS1_6B9_0: USINT;
	// Not USED Spare
	gu8_OrionBMS1_6B9_1: USINT;
	// Not USED Spare
	gu8_OrionBMS1_6B9_2: USINT;
	gu8_OrionBMS1_6B9_3: USINT;
	gu8_OrionBMS1_6B9_4: USINT;
	// Not USED Spare
	gu8_OrionBMS1_6B9_5: USINT;
	gu8_OrionBMS1_6B9_6: USINT;
	gu8_OrionBMS1_6B9_7: USINT;
	// 6BA Not USED Spare
	gu8_OrionBMS1_6BA_0: USINT;
	gu8_OrionBMS1_6BA_1: USINT;
	gu8_OrionBMS1_6BA_2: USINT;
	gu8_OrionBMS1_6BA_3: USINT;
	gu8_OrionBMS1_6BA_4: USINT;
	// Not USED Spare
	gu8_OrionBMS1_6BA_5: USINT;
	gu8_OrionBMS1_6BA_6: USINT;
	gu8_OrionBMS1_6BA_7: USINT;
	// 6BB Not USED Spare
	gu8_OrionBMS1_6BB_0: USINT;
	gu8_OrionBMS1_6BB_1: USINT;
	gu8_OrionBMS1_6BB_2: USINT;
	gu8_OrionBMS1_6BB_3: USINT;
	gu8_OrionBMS1_6BB_4: USINT;
	gu8_OrionBMS1_6BB_5: USINT;
	gu8_OrionBMS1_6BB_6: USINT;
	gu8_OrionBMS1_6BB_7: USINT;
	// 6BC Not USED Spare
	gu8_OrionBMS1_6BC_0: USINT;
	gu8_OrionBMS1_6BC_1: USINT;
	gu8_OrionBMS1_6BC_2: USINT;
	gu8_OrionBMS1_6BC_3: USINT;
	gu8_OrionBMS1_6BC_4: USINT;
	gu8_OrionBMS1_6BC_5: USINT;
	gu8_OrionBMS1_6BC_6: USINT;
	gu8_OrionBMS1_6BC_7: USINT;
	// 6BD Not USED Spare
	gu8_OrionBMS1_6BD_0: USINT;
	gu8_OrionBMS1_6BD_1: USINT;
	gu8_OrionBMS1_6BD_2: USINT;
	gu8_OrionBMS1_6BD_3: USINT;
	gu8_OrionBMS1_6BD_4: USINT;
	gu8_OrionBMS1_6BD_5: USINT;
	gu8_OrionBMS1_6BD_6: USINT;
	gu8_OrionBMS1_6BD_7: USINT;
	
	
	
	(**********************************************************)
	(*Rx Conversion*)
	gr_OrionBMS1_PackVoltage			:REAL;
	gr_OrionBMS1_PackCurrent			:REAL;
	gr_OrionBMS1_PackSOC				:REAL;
	gr_OrionBMS1_Max_Charging_Voltage	:REAL;
	
	
	(*DTC1 Flags*)
	OrionBMS1_DTCFlag1_0A07_DischargeLimitEnforcementFault1		:	BOOL;
	OrionBMS1_DTCFlag1_0A08_ChargerSafetyRelayFault1 			:	BOOL;
	OrionBMS1_DTCFlag1_0A09_InternalHardwareFault1				:	BOOL;
	OrionBMS1_DTCFlag1_0A0A_InternalHeatskinkThermistorFault 	:	BOOL;
	OrionBMS1_DTCFlag1_0A0B_InternalSoftwareFault1				:	BOOL;
	OrionBMS1_DTCFlag1_0A0C_HighestCellVoltageTooHighFault1 	:	BOOL;
	OrionBMS1_DTCFlag1_0A0E_LowestCellVoltageTooLowFault 		:	BOOL;
	OrionBMS1_DTCFlag1_0A10_PackTooHotFault1 					:	BOOL;
	OrionBMS1_DTCFlags_Reserved_Bit8 							:	BOOL;
	OrionBMS1_DTCFlags_Reserved_Bit9 							:	BOOL;
	OrionBMS1_DTCFlags_Reserved_Bit10 							:	BOOL;
	OrionBMS1_DTCFlags_Reserved_Bit11 							:	BOOL;
	OrionBMS1_DTCFlags_Reserved_Bit12 							:	BOOL;
	OrionBMS1_DTCFlags_Reserved_Bit13 							:	BOOL;
	OrionBMS1_DTCFlags_Reserved_Bit14 							:	BOOL;
	OrionBMS1_DTCFlags_Reserved_Bit15							:	BOOL;
	(*DTC2 Flags*)
	OrionBMS1_DTCFlags2_0A1F_InternalCommunicationFault			:	BOOL;
	OrionBMS1_DTCFlags2_0A12_CellBalancingStruckOffFault		:	BOOL;
	OrionBMS1_DTCFlags2_0A80_WeakCellFault						:	BOOL;
	OrionBMS1_DTCFlags2_0AFA_LowCellVoltageFault				:	BOOL;
	OrionBMS1_DTCFlags2_0A04_OpenWiringFault					:	BOOL;
	OrionBMS1_DTCFlags2_0AC0_CurrentSensorFault					:	BOOL;
	OrionBMS1_DTCFlags2_0A0D_HighestCellVoltageOver5vFault		:	BOOL;
	OrionBMS1_DTCFlags2_0A0F_CellASICFault						:	BOOL;
	OrionBMS1_DTCFlags2_0A02_WeakPackFault						:	BOOL;
	OrionBMS1_DTCFlags2_0A81_FanMonitorFault					:	BOOL;
	OrionBMS1_DTCFlags2_0A9C_ThermistorFault					:	BOOL;
	OrionBMS1_DTCFlags2_0100_ExternalCommunicationFault			:	BOOL;
	OrionBMS1_DTCFlags2_0560_RedundantPowerSupplyFault			:	BOOL;
	OrionBMS1_DTCFlags2_0AA6_HighVoltageIsolatonFault			:	BOOL;
	OrionBMS1_DTCFlags2_0A05_InputPowerSupplyFault				:	BOOL;
	OrionBMS1_DTCFlags2_0A06_ChargeLimitEnforcementFault		:	BOOL;
	
	(**********************************************************************)
	
	(* Custom Flag *)
	gq_BMS1_BalActive			:BOOL;
	gq_BMS1_Flag_1				:BOOL;
	gq_BMS1_Flag_2				:BOOL;
	gq_BMS1_Flag_3				:BOOL;
	gq_BMS1_Flag_4				:BOOL;
	gq_BMS1_Flag_5				:BOOL;
	gq_BMS1_Flag_6				:BOOL;
	gq_BMS1_Flag_7				:BOOL;
	
	(********************************************************************)
	(* Current Limit Flags *)
	
	
	
	gq_OrionBMS1_CommsLoss										:	BOOL;
	
	// Tx
	gu8_BMS1_MPO_1_State					: USINT;
	// Not connected to Anything. But it's Here.
	gu8_BMS1_MPO_2_State					: USINT;
	// Tx
	gu8_BMS1_MPO_3_State					: USINT;
	// Tx
	gu8_BMS1_MPO_4_State					: USINT;
	// Tx
	gu8_BMS1_MPE_State					: USINT;
END_VAR

// Application/CodeTemplate/POUs/PLC_PRG
///Tool version       : '6.5.7390.16348'
///Xml version        : '5.0.44'
///Control Unit       : 'VMU'
///Control Unit Type  : '5050'
///Export Time        : '29.06.2020 13:29.57'
///Export Path        : 'C:\Users\MatthewJoy\Desktop\Github Repository\P2030_Electra_VMU\P2101_Electra_VMU\VMUProject\VMU'
///Project File       : 'C:\Users\MatthewJoy\Desktop\Github Repository\P2030_Electra_VMU\P2101_Electra_VMU\VMUProject\VMUProject.net'
///Libraries Path     : 'C:\Users\MatthewJoy\Desktop\Github Repository\P2030_Electra_VMU\P2101_Electra_VMU\VMUProject\VMU\Libraries'
PROGRAM PLC_PRG

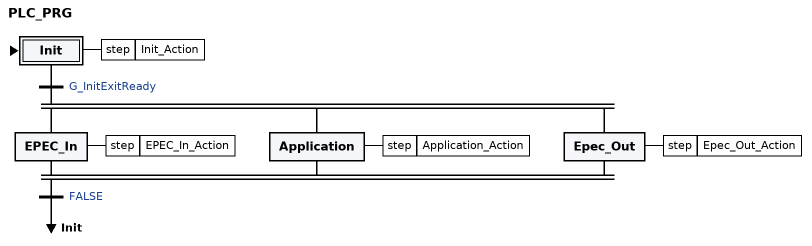
INITIAL_STEP Init:
    Init_Action(N);  // step action
END_STEP
TRANSITION FROM Init TO (EPEC_In, Application, Epec_Out)
    := G_InitExitReady;
END_TRANSITION
STEP EPEC_In:
    EPEC_In_Action(N);  // step action
END_STEP
STEP Application:
    Application_Action(N);  // step action
END_STEP
STEP Epec_Out:
    Epec_Out_Action(N);  // step action
END_STEP
TRANSITION FROM (EPEC_In, Application, Epec_Out) TO Init
    := FALSE;
END_TRANSITION
// branch label MainLoop

ACTION Application_Action:
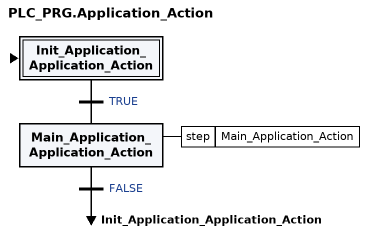
INITIAL_STEP Init_Application_Application_Action:
END_STEP
TRANSITION FROM Init_Application_Application_Action TO Main_Application_Application_Action
    := TRUE;
END_TRANSITION
STEP Main_Application_Application_Action:
    Main_Application_Action(N);  // step action
END_STEP
TRANSITION FROM Main_Application_Application_Action TO Init_Application_Application_Action
    := FALSE;
END_TRANSITION
END_ACTION

ACTION Bus_Action:


G_CAN1_Channel.CheckMessages();
G_CAN2_Channel.CheckMessages();
G_CAN3_Channel.CheckMessages();
G_CAN4_Channel.CheckMessages();

(* Update callback data *)
IF G_CAN1_Channel.GetLatestError() <> DWORD#0 THEN
	G_CANopen_CAN1_VAR.Callback_Error := EPEC_CANopen.Errors.CallbackError;
ELSE
	G_CANopen_CAN1_VAR.Callback_Error := EPEC_CANopen.Errors.NoError;
END_IF

(* Update protocol data *)
G_CANopen_CAN1.HB_Handler.Update(
	i_Enable := TRUE,
	o_Error => G_CANopen_CAN1_VAR.HB_Error
);
G_CANopen_CAN1.NMT_Handler.Update(
	i_Enable := TRUE,
	o_Error => G_CANopen_CAN1_VAR.NMT_Error
);
G_CANopen_CAN1.SSDO_Handler.Update(
	i_Enable := TRUE,
	o_Error => G_CANopen_CAN1_VAR.SSDO_Error
);
G_CANopen_CAN1.GFC_Handler.Update(
	i_Enable := TRUE,
	o_Error => G_CANopen_CAN1_VAR.GFC_Error
);

IF G_CANopen_CAN1_VAR.HB_Error = EPEC_CANopen.Errors.NoError AND
	G_CANopen_CAN1_VAR.NMT_Error = EPEC_CANopen.Errors.NoError AND
	G_CANopen_CAN1_VAR.SSDO_Error = EPEC_CANopen.Errors.NoError AND
	G_CANopen_CAN1_VAR.GFC_Error = EPEC_CANopen.Errors.NoError
THEN
	G_CANopenCan1ProtocolError := FALSE;
ELSE
	G_CANopenCan1ProtocolError := TRUE;
END_IF


(* Update callback data *)
IF G_CAN2_Channel.GetLatestError() <> DWORD#0 THEN
	G_CANopen_CAN2_VAR.Callback_Error := EPEC_CANopen.Errors.CallbackError;
ELSE
	G_CANopen_CAN2_VAR.Callback_Error := EPEC_CANopen.Errors.NoError;
END_IF

(* Update protocol data *)
G_CANopen_CAN2.HB_Handler.Update(
	i_Enable := TRUE,
	o_Error => G_CANopen_CAN2_VAR.HB_Error
);
G_CANopen_CAN2.NMT_Handler.Update(
	i_Enable := TRUE,
	o_Error => G_CANopen_CAN2_VAR.NMT_Error
);
G_CANopen_CAN2.SSDO_Handler.Update(
	i_Enable := TRUE,
	o_Error => G_CANopen_CAN2_VAR.SSDO_Error
);
G_CANopen_CAN2.GFC_Handler.Update(
	i_Enable := TRUE,
	o_Error => G_CANopen_CAN2_VAR.GFC_Error
);

IF G_CANopen_CAN2_VAR.HB_Error = EPEC_CANopen.Errors.NoError AND
	G_CANopen_CAN2_VAR.NMT_Error = EPEC_CANopen.Errors.NoError AND
	G_CANopen_CAN2_VAR.SSDO_Error = EPEC_CANopen.Errors.NoError AND
	G_CANopen_CAN2_VAR.GFC_Error = EPEC_CANopen.Errors.NoError
THEN
	G_CANopenCan2ProtocolError := FALSE;
ELSE
	G_CANopenCan2ProtocolError := TRUE;
END_IF


(* Update callback data *)
IF G_CAN3_Channel.GetLatestError() <> DWORD#0 THEN
	G_CANopen_CAN3_VAR.Callback_Error := EPEC_CANopen.Errors.CallbackError;
ELSE
	G_CANopen_CAN3_VAR.Callback_Error := EPEC_CANopen.Errors.NoError;
END_IF

(* Update protocol data *)
G_CANopen_CAN3.HB_Handler.Update(
	i_Enable := TRUE,
	o_Error => G_CANopen_CAN3_VAR.HB_Error
);
G_CANopen_CAN3.NMT_Handler.Update(
	i_Enable := TRUE,
	o_Error => G_CANopen_CAN3_VAR.NMT_Error
);
G_CANopen_CAN3.SSDO_Handler.Update(
	i_Enable := TRUE,
	o_Error => G_CANopen_CAN3_VAR.SSDO_Error
);
G_CANopen_CAN3.GFC_Handler.Update(
	i_Enable := TRUE,
	o_Error => G_CANopen_CAN3_VAR.GFC_Error
);

IF G_CANopen_CAN3_VAR.HB_Error = EPEC_CANopen.Errors.NoError AND
	G_CANopen_CAN3_VAR.NMT_Error = EPEC_CANopen.Errors.NoError AND
	G_CANopen_CAN3_VAR.SSDO_Error = EPEC_CANopen.Errors.NoError AND
	G_CANopen_CAN3_VAR.GFC_Error = EPEC_CANopen.Errors.NoError
THEN
	G_CANopenCan3ProtocolError := FALSE;
ELSE
	G_CANopenCan3ProtocolError := TRUE;
END_IF


(* Update callback data *)
IF G_CAN4_Channel.GetLatestError() <> DWORD#0 THEN
	G_CANopen_CAN4_VAR.Callback_Error := EPEC_CANopen.Errors.CallbackError;
ELSE
	G_CANopen_CAN4_VAR.Callback_Error := EPEC_CANopen.Errors.NoError;
END_IF

(* Update protocol data *)
G_CANopen_CAN4.HB_Handler.Update(
	i_Enable := TRUE,
	o_Error => G_CANopen_CAN4_VAR.HB_Error
);
G_CANopen_CAN4.NMT_Handler.Update(
	i_Enable := TRUE,
	o_Error => G_CANopen_CAN4_VAR.NMT_Error
);
G_CANopen_CAN4.SSDO_Handler.Update(
	i_Enable := TRUE,
	o_Error => G_CANopen_CAN4_VAR.SSDO_Error
);
G_CANopen_CAN4.GFC_Handler.Update(
	i_Enable := TRUE,
	o_Error => G_CANopen_CAN4_VAR.GFC_Error
);

IF G_CANopen_CAN4_VAR.HB_Error = EPEC_CANopen.Errors.NoError AND
	G_CANopen_CAN4_VAR.NMT_Error = EPEC_CANopen.Errors.NoError AND
	G_CANopen_CAN4_VAR.SSDO_Error = EPEC_CANopen.Errors.NoError AND
	G_CANopen_CAN4_VAR.GFC_Error = EPEC_CANopen.Errors.NoError
THEN
	G_CANopenCan4ProtocolError := FALSE;
ELSE
	G_CANopenCan4ProtocolError := TRUE;
END_IF


(*Check for nmt reset *)
IF G_CANopen_CAN1.NMT.StateChanged THEN
	IF G_CANopen_CAN1.NMT.LastNmtCommand = EPEC_CANopen.NMTCommand.Reset OR 
	   G_CANopen_CAN1.NMT.LastNmtCommand = EPEC_CANopen.NMTCommand.ResetCommunication 
	THEN
		(* If there is NMT reset command for IEC application CANopen device,
			IEC application is started after IEC cycle in execution. *)
		G_RESET_MODULE := TRUE;
	END_IF
END_IF

(*Check for nmt reset *)
IF G_CANopen_CAN2.NMT.StateChanged THEN
	IF G_CANopen_CAN2.NMT.LastNmtCommand = EPEC_CANopen.NMTCommand.Reset OR 
	   G_CANopen_CAN2.NMT.LastNmtCommand = EPEC_CANopen.NMTCommand.ResetCommunication 
	THEN
		(* If there is NMT reset command for IEC application CANopen device,
			IEC application is started after IEC cycle in execution. *)
		G_RESET_MODULE := TRUE;
	END_IF
END_IF

(*Check for nmt reset *)
IF G_CANopen_CAN3.NMT.StateChanged THEN
	IF G_CANopen_CAN3.NMT.LastNmtCommand = EPEC_CANopen.NMTCommand.Reset OR 
	   G_CANopen_CAN3.NMT.LastNmtCommand = EPEC_CANopen.NMTCommand.ResetCommunication 
	THEN
		(* If there is NMT reset command for IEC application CANopen device,
			IEC application is started after IEC cycle in execution. *)
		G_RESET_MODULE := TRUE;
	END_IF
END_IF

(*Check for nmt reset *)
IF G_CANopen_CAN4.NMT.StateChanged THEN
	IF G_CANopen_CAN4.NMT.LastNmtCommand = EPEC_CANopen.NMTCommand.Reset OR 
	   G_CANopen_CAN4.NMT.LastNmtCommand = EPEC_CANopen.NMTCommand.ResetCommunication 
	THEN
		(* If there is NMT reset command for IEC application CANopen device,
			IEC application is started after IEC cycle in execution. *)
		G_RESET_MODULE := TRUE;
	END_IF
END_IF



J1939_FB_CAN1(i_CANChannel:=G_CAN1_Channel,
	i_pRxPGNs:=ADR(J1939_CAN1.In.PGNs),
	i_NumberOfRxPGNs:=3,
	i_pTxPGNs:=0,
	i_NumberOfTxPGNs:=0);
J1939_FB_CAN4(i_CANChannel:=G_CAN4_Channel,
	i_pRxPGNs:=ADR(J1939_CAN4.In.PGNs),
	i_NumberOfRxPGNs:=3,
	i_pTxPGNs:=0,
	i_NumberOfTxPGNs:=0);
END_ACTION

ACTION Diag_Action:

(* Update functionalities for IO*)
	(* HW diagnostic *)
	AI_SupplyLogic := AI_MeanValue(AI_ARR_INDEX,ADR(AI_ARR_SupplyLogic[1]),1,50, 10); (* Filter logic supply raw values*)
	AI_Ref5V := AI_MeanValue(AI_ARR_INDEX,ADR(AI_ARR_Ref5V[1]),1,50, 10); (* Filter 5V ref raw values. *)
	AI_Ref10V := AI_MeanValue(AI_ARR_INDEX,ADR(AI_ARR_Ref10V[1]),1,50, 10); (* Filter 10V ref raw values. *)
	AI_PCBTemperature := AI_MeanValue(AI_ARR_INDEX,ADR(AI_ARR_PCBTemperature[1]), 1,50, 10);
	AI_SupplyPower1 := AI_MeanValue(AI_ARR_INDEX,ADR(AI_ARR_SupplyPower1[1]), 1,50, 10); (* Filter power switch 1 raw values*)
	AI_SupplyPower2 := AI_MeanValue(AI_ARR_INDEX,ADR(AI_ARR_SupplyPower2[1]), 1,50, 10); (* Filter power switch 2 raw values*)
	AI_10VPullUpSupply := AI_MeanValue(AI_ARR_INDEX,ADR(AI_ARR_10VPullUpSupply[1]),1,50, 10);
	AI_InternADCReference := AI_MeanValue(AI_ARR_INDEX,ADR(AI_ARR_InternADCReference[1]), 1,50, 10);
	AI_CoreTemperature := AI_MeanValue(AI_ARR_INDEX,ADR(AI_ARR_CoreTemperature[1]), 1,50, 10);
	AI_Power1Pin := AI_MeanValue(AI_ARR_INDEX,ADR(AI_ARR_Power1Pin [1]), 1,50, 10);
	AI_Power2Pin := AI_MeanValue(AI_ARR_INDEX,ADR(AI_ARR_Power2Pin [1]), 1,50, 10);

	G_HWDiagnostics(
		i_SupplyVoltage1:=AI_SupplyLogic,
		i_SupplyVoltage2:=AI_Power1Pin ,
		i_SupplyVoltage3:=AI_Power2Pin,
		i_Ref5V:=AI_Ref5V,
		i_Ref10V:=AI_Ref10V,
		i_Pullup10V := AI_10VPullUpSupply,
		i_RefADC := AI_InternADCReference,
		i_Temperature1 := AI_CoreTemperature,
		i_Temperature2 := AI_PCBTemperature,
		i_SupplyVoltageHighLimit := INT_TO_UINT(G_SupplyVoltageHighLimit),
		i_SupplyVoltageLowLimit := INT_TO_UINT(G_SupplyVoltageLowLimit),
		i_Ref5VHighLimit := INT_TO_UINT(G_Ref5VHighLimit),
		i_Ref5VLowLimit := INT_TO_UINT(G_Ref5VLowLimit),
		i_Ref10VHighLimit := INT_TO_UINT(G_Ref10VHighLimit),
		i_Ref10VLowLimit := INT_TO_UINT(G_Ref10VLowLimit),
		i_PullUp10VHighLimit := INT_TO_UINT(G_PullUp10VHighLimit),
		i_PullUp10VLowLimit := INT_TO_UINT(G_PullUp10VLowLimit),
		i_RefADCVHighLimit := INT_TO_UINT(G_RefADCVHighLimit),
		i_RefADCVLowLimit := INT_TO_UINT(G_RefADCVLowLimit),
		i_TempHighLimit := G_TempHighLimit,
		i_TempLowLimit := G_TempLowLimit,
		i_CycleTimeHighLimit := INT_TO_UINT(G_CycleTimeHighLimit));

		SUPPLY_Logic := G_HWDiagnostics.o_SupplyVoltage1;
		SUPPLY_Power1Pin:= G_HWDiagnostics.o_SupplyVoltage2;
		SUPPLY_Power2Pin := G_HWDiagnostics.o_SupplyVoltage3;
		REF_10V := G_HWDiagnostics.o_Ref10V;
		REF_5V := G_HWDiagnostics.o_Ref5V;
		REF_10VPullUpSupply := G_HWDiagnostics.o_PullUp10V;
		REF_InternADC := G_HWDiagnostics.o_RefADCV;
		TEMP_PCB := G_HWDiagnostics.o_Temperature2;
		TEMP_CoreTemperature := G_HWDiagnostics.o_Temperature1;

		SUPPLY_Power1 := ADC_To_mAorV(AI_SupplyPower1,G_AIType.Supply);
		SUPPLY_Power2 := ADC_To_mAorV(AI_SupplyPower2,G_AIType.Supply);


	(* Update power switches and scale voltages measurement *)
		SYSTEM_PWR_SWT_SET_STATE(0,BOOL_TO_BYTE(POWER_1_Enable));
	(* Update power switches *)
		SYSTEM_PWR_SWT_SET_STATE(1,BOOL_TO_BYTE(POWER_2_Enable));









(*########################################################*)
(*This block is created implicit. Don't add own code here.*)
(*########################################################*)

(* Diagnostics for CAN interfaces *)





(* CANopen networks management and diagnostics  *)





(* System Ok conditions *)
G_SystemOk:=NOT(G_HWDiagnostics.o_Temperature1High) AND
		NOT(G_HWDiagnostics.o_Temperature1Low) AND
		NOT(G_HWDiagnostics.o_Temperature2High) AND
		NOT(G_HWDiagnostics.o_Temperature2Low) AND
		NOT(G_HWDiagnostics.o_SupplyVoltage1High) AND
		NOT(G_HWDiagnostics.o_SupplyVoltage1Low) AND
		NOT(G_HWDiagnostics.o_PullUp10VHigh) AND
		NOT(G_HWDiagnostics.o_PullUp10VLow) AND
		NOT(G_HWDiagnostics.o_RefADCVHigh) AND
		NOT(G_HWDiagnostics.o_RefADCVLow) AND
		NOT (ERR_FLAG_IO_INIT);



POWER_1_Enable:=G_SystemOk;
POWER_2_Enable:=G_SystemOk;



IO_SET_LED(i_SystemOk:=G_SystemOk, i_RunWithErrors:=G_ActiveError, i_InitState:=NOT(G_InitExitReady));

IF G_HWDiagnostics.o_SupplyVoltage1 > G_LowLimitForParameterSaving THEN
	G_Common.ParHandler.DisableChanges(i_DisableChanges := FALSE);
ELSE
	G_Common.ParHandler.DisableChanges(i_DisableChanges := TRUE);
END_IF
END_ACTION

ACTION EPEC_In_Action:
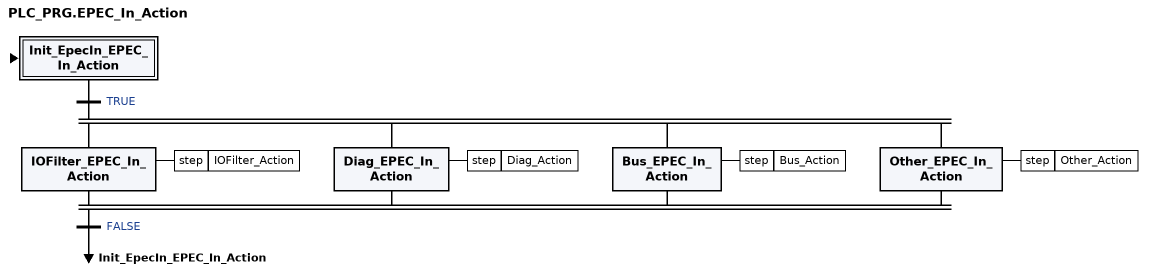
INITIAL_STEP Init_EpecIn_EPEC_In_Action:
END_STEP
TRANSITION FROM Init_EpecIn_EPEC_In_Action TO (IOFilter_EPEC_In_Action, Diag_EPEC_In_Action, Bus_EPEC_In_Action, Other_EPEC_In_Action)
    := TRUE;
END_TRANSITION
STEP IOFilter_EPEC_In_Action:
    IOFilter_Action(N);  // step action
END_STEP
STEP Diag_EPEC_In_Action:
    Diag_Action(N);  // step action
END_STEP
STEP Bus_EPEC_In_Action:
    Bus_Action(N);  // step action
END_STEP
STEP Other_EPEC_In_Action:
    Other_Action(N);  // step action
END_STEP
TRANSITION FROM (IOFilter_EPEC_In_Action, Diag_EPEC_In_Action, Bus_EPEC_In_Action, Other_EPEC_In_Action) TO Init_EpecIn_EPEC_In_Action
    := FALSE;
END_TRANSITION
// branch label EpecInMainLoop
END_ACTION

ACTION Epec_Out_Action:
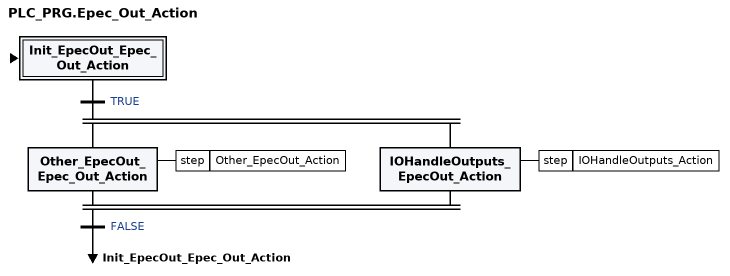
INITIAL_STEP Init_EpecOut_Epec_Out_Action:
END_STEP
TRANSITION FROM Init_EpecOut_Epec_Out_Action TO (Other_EpecOut_Epec_Out_Action, IOHandleOutputs_EpecOut_Action)
    := TRUE;
END_TRANSITION
STEP Other_EpecOut_Epec_Out_Action:
    Other_EpecOut_Action(N);  // step action
END_STEP
STEP IOHandleOutputs_EpecOut_Action:
    IOHandleOutputs_Action(N);  // step action
END_STEP
TRANSITION FROM (Other_EpecOut_Epec_Out_Action, IOHandleOutputs_EpecOut_Action) TO Init_EpecOut_Epec_Out_Action
    := FALSE;
END_TRANSITION
// branch label EpecOutMainLoop
END_ACTION

ACTION Init_Action:
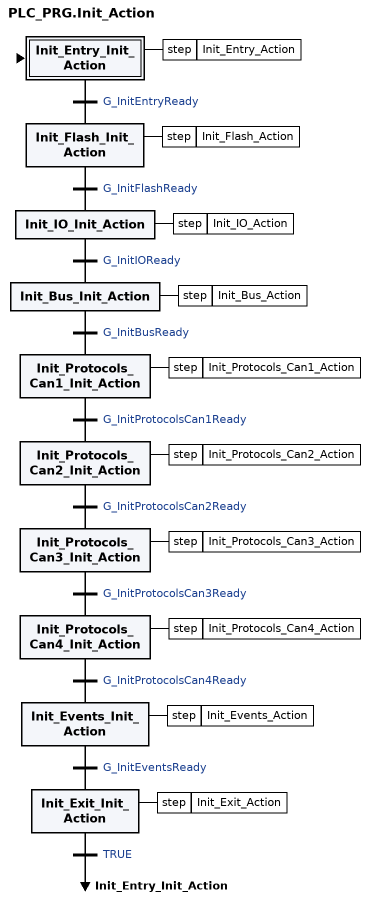
INITIAL_STEP Init_Entry_Init_Action:
    Init_Entry_Action(N);  // step action
END_STEP
TRANSITION FROM Init_Entry_Init_Action TO Init_Flash_Init_Action
    := G_InitEntryReady;
END_TRANSITION
STEP Init_Flash_Init_Action:
    Init_Flash_Action(N);  // step action
END_STEP
TRANSITION FROM Init_Flash_Init_Action TO Init_IO_Init_Action
    := G_InitFlashReady;
END_TRANSITION
STEP Init_IO_Init_Action:
    Init_IO_Action(N);  // step action
END_STEP
TRANSITION FROM Init_IO_Init_Action TO Init_Bus_Init_Action
    := G_InitIOReady;
END_TRANSITION
STEP Init_Bus_Init_Action:
    Init_Bus_Action(N);  // step action
END_STEP
TRANSITION FROM Init_Bus_Init_Action TO Init_Protocols_Can1_Init_Action
    := G_InitBusReady;
END_TRANSITION
STEP Init_Protocols_Can1_Init_Action:
    Init_Protocols_Can1_Action(N);  // step action
END_STEP
TRANSITION FROM Init_Protocols_Can1_Init_Action TO Init_Protocols_Can2_Init_Action
    := G_InitProtocolsCan1Ready;
END_TRANSITION
STEP Init_Protocols_Can2_Init_Action:
    Init_Protocols_Can2_Action(N);  // step action
END_STEP
TRANSITION FROM Init_Protocols_Can2_Init_Action TO Init_Protocols_Can3_Init_Action
    := G_InitProtocolsCan2Ready;
END_TRANSITION
STEP Init_Protocols_Can3_Init_Action:
    Init_Protocols_Can3_Action(N);  // step action
END_STEP
TRANSITION FROM Init_Protocols_Can3_Init_Action TO Init_Protocols_Can4_Init_Action
    := G_InitProtocolsCan3Ready;
END_TRANSITION
STEP Init_Protocols_Can4_Init_Action:
    Init_Protocols_Can4_Action(N);  // step action
END_STEP
TRANSITION FROM Init_Protocols_Can4_Init_Action TO Init_Events_Init_Action
    := G_InitProtocolsCan4Ready;
END_TRANSITION
STEP Init_Events_Init_Action:
    Init_Events_Action(N);  // step action
END_STEP
TRANSITION FROM Init_Events_Init_Action TO Init_Exit_Init_Action
    := G_InitEventsReady;
END_TRANSITION
STEP Init_Exit_Init_Action:
    Init_Exit_Action(N);  // step action
END_STEP
TRANSITION FROM Init_Exit_Init_Action TO Init_Entry_Init_Action
    := TRUE;
END_TRANSITION
END_ACTION

ACTION Init_Bus_Action:
(*###########################################################*)
(*This block is created implicit. Don't add own code to here.*)
(*###########################################################*)

G_CAN1_Channel.InitCAN(i_Channel:=0, i_BitRate:=G_SystemInfo.CAN1_Comms[3], i_Flags:=0);

G_CAN2_Channel.InitCAN(i_Channel:=1, i_BitRate:=G_SystemInfo.CAN2_Comms[3], i_Flags:=0);

G_CAN3_Channel.InitCAN(i_Channel:=2, i_BitRate:=G_SystemInfo.CAN3_Comms[3], i_Flags:=0);

G_CAN4_Channel.InitCAN(i_Channel:=3, i_BitRate:=G_SystemInfo.CAN4_Comms[3], i_Flags:=0);


G_InitBusReady := TRUE;
END_ACTION

ACTION Init_Entry_Action:
(*###########################################################*)
(*This block is created implicit. Don't add own code to here.*)
(*###########################################################*)
/// Call user init until flag is set on.
MainInit();
G_InitEntryReady := MainInit.o_MainInitReady;

IF TRUE = G_InitEntryReady THEN




    CmpApp.AppGetProjectInformation(pApp:=CmpApp.AppGetCurrent(ADR(G_FunctionResult)),pInfo:=ADR(G_SystemInfo.ProjectInfo));
    (* Read system parameters from flash *) 
    SystemParameters.ReadData(); 
  
